  PROC DrawPart231()
    MoveL Offs(pOrigin,236.82,333.03,0.00),v40,z0,tPen\WObj:=wPaper;
    MoveL Offs(pOrigin,238.31,333.31,0.00),v40,z0,tPen\WObj:=wPaper;
    MoveL Offs(pOrigin,238.10,333.91,0.00),v40,z0,tPen\WObj:=wPaper;
    MoveL Offs(pOrigin,233.85,333.91,0.00),v40,z0,tPen\WObj:=wPaper;
    MoveL Offs(pOrigin,233.47,333.82,0.00),v40,z0,tPen\WObj:=wPaper;
    MoveL Offs(pOrigin,235.43,335.78,0.00),v40,z0,tPen\WObj:=wPaper;
    MoveL Offs(pOrigin,236.39,335.84,0.00),v40,z0,tPen\WObj:=wPaper;
    MoveL Offs(pOrigin,241.65,330.58,0.00),v40,z0,tPen\WObj:=wPaper;
    MoveL Offs(pOrigin,240.80,330.70,0.00),v40,z0,tPen\WObj:=wPaper;
    MoveL Offs(pOrigin,239.45,329.35,0.00),v40,z0,tPen\WObj:=wPaper;
    MoveL Offs(pOrigin,239.38,330.12,0.00),v40,z0,tPen\WObj:=wPaper;
    MoveL Offs(pOrigin,239.16,331.40,0.00),v40,z0,tPen\WObj:=wPaper;
    MoveL Offs(pOrigin,239.59,332.04,0.00),v40,z0,tPen\WObj:=wPaper;
    MoveL Offs(pOrigin,239.91,332.80,0.00),v40,z0,tPen\WObj:=wPaper;
    MoveL Offs(pOrigin,238.71,331.59,0.00),v40,z0,tPen\WObj:=wPaper;
    MoveL Offs(pOrigin,239.31,330.70,0.00),v40,z0,tPen\WObj:=wPaper;
    MoveL Offs(pOrigin,240.51,331.90,0.00),v40,fine,tPen\WObj:=wPaper;
    MoveL Offs(pOrigin,240.51,331.90,6.00),v60,z5,tPen\WObj:=wPaper;
    MoveL Offs(pOrigin,240.44,330.12,6.00),vTravel,z5,tPen\WObj:=wPaper;
    MoveL Offs(pOrigin,240.44,330.12,0.00),v60,z0,tPen\WObj:=wPaper;
    MoveL Offs(pOrigin,240.23,328.00,0.00),v40,z0,tPen\WObj:=wPaper;
    MoveL Offs(pOrigin,240.23,328.00,0.00),v40,z0,tPen\WObj:=wPaper;
    MoveL Offs(pOrigin,240.44,328.00,0.00),v40,z0,tPen\WObj:=wPaper;
    MoveL Offs(pOrigin,239.80,326.30,0.00),v40,z0,tPen\WObj:=wPaper;
    MoveL Offs(pOrigin,239.80,326.73,0.00),v40,z0,tPen\WObj:=wPaper;
    MoveL Offs(pOrigin,239.16,327.15,0.00),v40,z0,tPen\WObj:=wPaper;
    MoveL Offs(pOrigin,239.38,328.00,0.00),v40,z0,tPen\WObj:=wPaper;
    MoveL Offs(pOrigin,239.38,328.00,0.00),v40,z0,tPen\WObj:=wPaper;
    MoveL Offs(pOrigin,239.38,330.12,0.00),v40,z0,tPen\WObj:=wPaper;
    MoveL Offs(pOrigin,239.38,330.12,0.00),v40,z0,tPen\WObj:=wPaper;
    MoveL Offs(pOrigin,240.44,330.12,0.00),v40,z0,tPen\WObj:=wPaper;
    MoveL Offs(pOrigin,241.10,329.50,0.00),v40,z0,tPen\WObj:=wPaper;
    MoveL Offs(pOrigin,220.51,308.92,0.00),v40,z0,tPen\WObj:=wPaper;
    MoveL Offs(pOrigin,220.68,309.09,0.00),v40,z0,tPen\WObj:=wPaper;
    MoveL Offs(pOrigin,218.76,309.51,0.00),v40,z0,tPen\WObj:=wPaper;
    MoveL Offs(pOrigin,218.05,310.01,0.00),v40,z0,tPen\WObj:=wPaper;
    MoveL Offs(pOrigin,218.05,311.35,0.00),v40,z0,tPen\WObj:=wPaper;
    MoveL Offs(pOrigin,216.85,311.57,0.00),v40,z0,tPen\WObj:=wPaper;
    MoveL Offs(pOrigin,217.06,310.36,0.00),v40,z0,tPen\WObj:=wPaper;
    MoveL Offs(pOrigin,218.05,310.01,0.00),v40,z0,tPen\WObj:=wPaper;
    MoveL Offs(pOrigin,217.55,310.15,0.00),v40,z0,tPen\WObj:=wPaper;
    MoveL Offs(pOrigin,217.55,315.68,0.00),v40,z0,tPen\WObj:=wPaper;
    MoveL Offs(pOrigin,217.28,315.96,0.00),v40,z0,tPen\WObj:=wPaper;
    MoveL Offs(pOrigin,231.51,315.96,0.00),v40,z0,tPen\WObj:=wPaper;
    MoveL Offs(pOrigin,231.28,316.95,0.00),v40,z0,tPen\WObj:=wPaper;
    MoveL Offs(pOrigin,231.28,322.05,0.00),v40,z0,tPen\WObj:=wPaper;
    MoveL Offs(pOrigin,232.33,322.05,0.00),v40,z0,tPen\WObj:=wPaper;
    MoveL Offs(pOrigin,232.33,318.44,0.00),v40,z0,tPen\WObj:=wPaper;
    MoveL Offs(pOrigin,232.57,318.44,0.00),v40,z0,tPen\WObj:=wPaper;
    MoveL Offs(pOrigin,231.94,319.08,0.00),v40,z0,tPen\WObj:=wPaper;
    MoveL Offs(pOrigin,231.09,319.08,0.00),v40,z0,tPen\WObj:=wPaper;
    MoveL Offs(pOrigin,231.09,319.08,0.00),v40,z0,tPen\WObj:=wPaper;
    MoveL Offs(pOrigin,231.16,320.56,0.00),v40,z0,tPen\WObj:=wPaper;
    MoveL Offs(pOrigin,233.43,323.11,0.00),v40,z0,tPen\WObj:=wPaper;
    MoveL Offs(pOrigin,233.21,322.69,0.00),v40,z0,tPen\WObj:=wPaper;
    MoveL Offs(pOrigin,233.43,323.11,0.00),v40,z0,tPen\WObj:=wPaper;
    MoveL Offs(pOrigin,233.21,322.69,0.00),v40,z0,tPen\WObj:=wPaper;
    MoveL Offs(pOrigin,233.39,322.26,0.00),v40,z0,tPen\WObj:=wPaper;
    MoveL Offs(pOrigin,233.39,319.71,0.00),v40,fine,tPen\WObj:=wPaper;
    MoveL Offs(pOrigin,233.39,319.71,6.00),v60,z5,tPen\WObj:=wPaper;
    MoveL Offs(pOrigin,234.27,320.56,6.00),vTravel,z5,tPen\WObj:=wPaper;
    MoveL Offs(pOrigin,234.27,320.56,0.00),v60,z0,tPen\WObj:=wPaper;
    MoveL Offs(pOrigin,234.27,320.14,0.00),v40,z0,tPen\WObj:=wPaper;
    MoveL Offs(pOrigin,232.79,318.44,0.00),v40,z0,tPen\WObj:=wPaper;
    MoveL Offs(pOrigin,232.79,318.44,0.00),v40,z0,tPen\WObj:=wPaper;
    MoveL Offs(pOrigin,233.21,317.16,0.00),v40,z0,tPen\WObj:=wPaper;
    MoveL Offs(pOrigin,232.57,315.25,0.00),v40,z0,tPen\WObj:=wPaper;
    MoveL Offs(pOrigin,232.57,313.12,0.00),v40,z0,tPen\WObj:=wPaper;
    MoveL Offs(pOrigin,233.21,311.99,0.00),v40,z0,tPen\WObj:=wPaper;
    MoveL Offs(pOrigin,233.64,312.49,0.00),v40,z0,tPen\WObj:=wPaper;
    MoveL Offs(pOrigin,233.43,313.34,0.00),v40,z0,tPen\WObj:=wPaper;
    MoveL Offs(pOrigin,233.64,315.25,0.00),v40,z0,tPen\WObj:=wPaper;
    MoveL Offs(pOrigin,234.20,316.95,0.00),v40,z0,tPen\WObj:=wPaper;
    MoveL Offs(pOrigin,235.34,317.80,0.00),v40,z0,tPen\WObj:=wPaper;
    MoveL Offs(pOrigin,237.04,320.77,0.00),v40,z0,tPen\WObj:=wPaper;
    MoveL Offs(pOrigin,237.04,320.77,0.00),v40,z0,tPen\WObj:=wPaper;
    MoveL Offs(pOrigin,238.10,321.84,0.00),v40,z0,tPen\WObj:=wPaper;
    MoveL Offs(pOrigin,237.61,322.26,0.00),v40,z0,tPen\WObj:=wPaper;
    MoveL Offs(pOrigin,237.61,324.18,0.00),v40,z0,tPen\WObj:=wPaper;
    MoveL Offs(pOrigin,236.56,323.96,0.00),v40,z0,tPen\WObj:=wPaper;
    MoveL Offs(pOrigin,236.56,321.41,0.00),v40,z0,tPen\WObj:=wPaper;
    MoveL Offs(pOrigin,235.55,321.41,0.00),v40,z0,tPen\WObj:=wPaper;
    MoveL Offs(pOrigin,234.91,320.70,0.00),v40,z0,tPen\WObj:=wPaper;
    MoveL Offs(pOrigin,234.35,320.77,0.00),v40,z0,tPen\WObj:=wPaper;
    MoveL Offs(pOrigin,234.70,321.84,0.00),v40,z0,tPen\WObj:=wPaper;
    MoveL Offs(pOrigin,235.55,322.05,0.00),v40,fine,tPen\WObj:=wPaper;
    MoveL Offs(pOrigin,235.55,322.05,6.00),v60,z5,tPen\WObj:=wPaper;
    MoveL Offs(pOrigin,235.50,320.77,6.00),vTravel,z5,tPen\WObj:=wPaper;
    MoveL Offs(pOrigin,235.50,320.77,0.00),v60,z0,tPen\WObj:=wPaper;
    MoveL Offs(pOrigin,235.50,323.54,0.00),v40,z0,tPen\WObj:=wPaper;
    MoveL Offs(pOrigin,236.19,324.41,0.00),v40,z0,tPen\WObj:=wPaper;
    MoveL Offs(pOrigin,239.59,324.41,0.00),v40,z0,tPen\WObj:=wPaper;
    MoveL Offs(pOrigin,240.03,323.96,0.00),v40,z0,tPen\WObj:=wPaper;
    MoveL Offs(pOrigin,226.66,310.58,0.00),v40,fine,tPen\WObj:=wPaper;
    MoveL Offs(pOrigin,226.66,310.58,6.00),v60,z5,tPen\WObj:=wPaper;
    MoveL Offs(pOrigin,226.62,313.85,6.00),vTravel,z5,tPen\WObj:=wPaper;
    MoveL Offs(pOrigin,226.62,313.85,0.00),v60,z0,tPen\WObj:=wPaper;
    MoveL Offs(pOrigin,216.00,313.85,0.00),v40,z0,tPen\WObj:=wPaper;
    MoveL Offs(pOrigin,215.57,313.55,0.00),v40,z0,tPen\WObj:=wPaper;
    MoveL Offs(pOrigin,215.15,313.98,0.00),v40,z0,tPen\WObj:=wPaper;
    MoveL Offs(pOrigin,215.15,314.61,0.00),v40,z0,tPen\WObj:=wPaper;
    MoveL Offs(pOrigin,214.94,313.85,0.00),v40,z0,tPen\WObj:=wPaper;
    MoveL Offs(pOrigin,213.24,313.85,0.00),v40,z0,tPen\WObj:=wPaper;
    MoveL Offs(pOrigin,212.81,314.40,0.00),v40,z0,tPen\WObj:=wPaper;
    MoveL Offs(pOrigin,212.60,314.83,0.00),v40,z0,tPen\WObj:=wPaper;
    MoveL Offs(pOrigin,212.81,314.40,0.00),v40,z0,tPen\WObj:=wPaper;
    MoveL Offs(pOrigin,212.81,314.90,0.00),v40,z0,tPen\WObj:=wPaper;
    MoveL Offs(pOrigin,214.30,314.90,0.00),v40,z0,tPen\WObj:=wPaper;
    MoveL Offs(pOrigin,213.88,315.96,0.00),v40,z0,tPen\WObj:=wPaper;
    MoveL Offs(pOrigin,212.60,315.96,0.00),v40,z0,tPen\WObj:=wPaper;
    MoveL Offs(pOrigin,211.96,315.67,0.00),v40,z0,tPen\WObj:=wPaper;
    MoveL Offs(pOrigin,212.88,314.61,0.00),v40,z0,tPen\WObj:=wPaper;
    MoveL Offs(pOrigin,213.24,313.55,0.00),v40,z0,tPen\WObj:=wPaper;
    MoveL Offs(pOrigin,213.02,313.12,0.00),v40,z0,tPen\WObj:=wPaper;
    MoveL Offs(pOrigin,212.18,312.79,0.00),v40,z0,tPen\WObj:=wPaper;
    MoveL Offs(pOrigin,224.08,312.79,0.00),v40,fine,tPen\WObj:=wPaper;
    MoveL Offs(pOrigin,224.08,312.79,6.00),v60,z5,tPen\WObj:=wPaper;
    MoveL Offs(pOrigin,224.94,314.40,6.00),vTravel,z5,tPen\WObj:=wPaper;
    MoveL Offs(pOrigin,224.94,314.40,0.00),v60,z0,tPen\WObj:=wPaper;
    MoveL Offs(pOrigin,224.94,319.92,0.00),v40,z0,tPen\WObj:=wPaper;
  ENDPROC

  PROC DrawPart232()
    MoveL Offs(pOrigin,223.89,320.35,0.00),v40,z0,tPen\WObj:=wPaper;
    MoveL Offs(pOrigin,223.89,315.68,0.00),v40,z0,tPen\WObj:=wPaper;
    MoveL Offs(pOrigin,224.29,316.10,0.00),v40,z0,tPen\WObj:=wPaper;
    MoveL Offs(pOrigin,224.07,314.61,0.00),v40,z0,tPen\WObj:=wPaper;
    MoveL Offs(pOrigin,224.64,313.76,0.00),v40,z0,tPen\WObj:=wPaper;
    MoveL Offs(pOrigin,224.64,312.49,0.00),v40,z0,tPen\WObj:=wPaper;
    MoveL Offs(pOrigin,225.42,310.79,0.00),v40,z0,tPen\WObj:=wPaper;
    MoveL Offs(pOrigin,227.48,310.65,0.00),v40,z0,tPen\WObj:=wPaper;
    MoveL Offs(pOrigin,226.84,313.12,0.00),v40,z0,tPen\WObj:=wPaper;
    MoveL Offs(pOrigin,226.84,314.40,0.00),v40,z0,tPen\WObj:=wPaper;
    MoveL Offs(pOrigin,228.54,318.23,0.00),v40,fine,tPen\WObj:=wPaper;
    MoveL Offs(pOrigin,228.54,318.23,6.00),v60,z5,tPen\WObj:=wPaper;
    MoveL Offs(pOrigin,228.96,316.74,6.00),vTravel,z5,tPen\WObj:=wPaper;
    MoveL Offs(pOrigin,228.96,316.74,0.00),v60,z0,tPen\WObj:=wPaper;
    MoveL Offs(pOrigin,229.81,316.74,0.00),v40,z0,tPen\WObj:=wPaper;
    MoveL Offs(pOrigin,230.66,318.01,0.00),v40,z0,tPen\WObj:=wPaper;
    MoveL Offs(pOrigin,230.66,318.01,0.00),v40,z0,tPen\WObj:=wPaper;
    MoveL Offs(pOrigin,231.09,319.08,0.00),v40,fine,tPen\WObj:=wPaper;
    MoveL Offs(pOrigin,231.09,319.08,6.00),v60,z5,tPen\WObj:=wPaper;
    MoveL Offs(pOrigin,231.30,317.80,6.00),vTravel,z5,tPen\WObj:=wPaper;
    MoveL Offs(pOrigin,231.30,317.80,0.00),v60,z0,tPen\WObj:=wPaper;
    MoveL Offs(pOrigin,231.94,317.80,0.00),v40,z0,tPen\WObj:=wPaper;
    MoveL Offs(pOrigin,232.57,318.44,0.00),v40,z0,tPen\WObj:=wPaper;
    MoveL Offs(pOrigin,232.79,318.44,0.00),v40,z0,tPen\WObj:=wPaper;
    MoveL Offs(pOrigin,232.15,317.80,0.00),v40,z0,tPen\WObj:=wPaper;
    MoveL Offs(pOrigin,232.15,317.80,0.00),v40,z0,tPen\WObj:=wPaper;
    MoveL Offs(pOrigin,231.51,314.61,0.00),v40,z0,tPen\WObj:=wPaper;
    MoveL Offs(pOrigin,230.88,313.76,0.00),v40,z0,tPen\WObj:=wPaper;
    MoveL Offs(pOrigin,230.88,313.76,0.00),v40,z0,tPen\WObj:=wPaper;
    MoveL Offs(pOrigin,230.80,312.27,0.00),v40,z0,tPen\WObj:=wPaper;
    MoveL Offs(pOrigin,229.25,312.91,0.00),v40,z0,tPen\WObj:=wPaper;
    MoveL Offs(pOrigin,228.96,316.74,0.00),v40,fine,tPen\WObj:=wPaper;
    MoveL Offs(pOrigin,228.96,316.74,6.00),v60,z5,tPen\WObj:=wPaper;
    MoveL Offs(pOrigin,230.45,316.10,6.00),vTravel,z5,tPen\WObj:=wPaper;
    MoveL Offs(pOrigin,230.45,316.10,0.00),v60,z0,tPen\WObj:=wPaper;
    MoveL Offs(pOrigin,230.45,314.19,0.00),v40,z0,tPen\WObj:=wPaper;
    MoveL Offs(pOrigin,230.88,313.76,0.00),v40,z0,tPen\WObj:=wPaper;
    MoveL Offs(pOrigin,230.88,313.85,0.00),v40,z0,tPen\WObj:=wPaper;
    MoveL Offs(pOrigin,227.90,313.85,0.00),v40,fine,tPen\WObj:=wPaper;
    MoveL Offs(pOrigin,227.90,313.85,6.00),v60,z5,tPen\WObj:=wPaper;
    MoveL Offs(pOrigin,229.17,315.04,6.00),vTravel,z5,tPen\WObj:=wPaper;
    MoveL Offs(pOrigin,229.17,315.04,0.00),v60,z0,tPen\WObj:=wPaper;
    MoveL Offs(pOrigin,229.17,321.62,0.00),v40,z0,tPen\WObj:=wPaper;
    MoveL Offs(pOrigin,229.39,322.30,0.00),v40,z0,tPen\WObj:=wPaper;
    MoveL Offs(pOrigin,247.66,322.30,0.00),v40,z0,tPen\WObj:=wPaper;
    MoveL Offs(pOrigin,248.17,321.41,0.00),v40,z0,tPen\WObj:=wPaper;
    MoveL Offs(pOrigin,248.17,319.29,0.00),v40,z0,tPen\WObj:=wPaper;
    MoveL Offs(pOrigin,248.94,319.08,0.00),v40,z0,tPen\WObj:=wPaper;
    MoveL Offs(pOrigin,249.79,318.65,0.00),v40,z0,tPen\WObj:=wPaper;
    MoveL Offs(pOrigin,249.79,318.65,0.00),v40,z0,tPen\WObj:=wPaper;
    MoveL Offs(pOrigin,249.50,317.16,0.00),v40,z0,tPen\WObj:=wPaper;
    MoveL Offs(pOrigin,248.02,315.89,0.00),v40,z0,tPen\WObj:=wPaper;
    MoveL Offs(pOrigin,247.17,313.12,0.00),v40,z0,tPen\WObj:=wPaper;
    MoveL Offs(pOrigin,246.81,312.84,0.00),v40,z0,tPen\WObj:=wPaper;
    MoveL Offs(pOrigin,246.39,313.34,0.00),v40,z0,tPen\WObj:=wPaper;
    MoveL Offs(pOrigin,246.39,314.40,0.00),v40,z0,tPen\WObj:=wPaper;
    MoveL Offs(pOrigin,247.02,317.16,0.00),v40,z0,tPen\WObj:=wPaper;
    MoveL Offs(pOrigin,247.02,317.16,0.00),v40,z0,tPen\WObj:=wPaper;
    MoveL Offs(pOrigin,247.45,318.86,0.00),v40,z0,tPen\WObj:=wPaper;
    MoveL Offs(pOrigin,247.45,318.86,0.00),v40,z0,tPen\WObj:=wPaper;
    MoveL Offs(pOrigin,245.75,318.44,0.00),v40,z0,tPen\WObj:=wPaper;
    MoveL Offs(pOrigin,244.05,318.44,0.00),v40,z0,tPen\WObj:=wPaper;
    MoveL Offs(pOrigin,244.05,318.44,0.00),v40,z0,tPen\WObj:=wPaper;
    MoveL Offs(pOrigin,244.26,319.50,0.00),v40,z0,tPen\WObj:=wPaper;
    MoveL Offs(pOrigin,245.11,320.56,0.00),v40,z0,tPen\WObj:=wPaper;
    MoveL Offs(pOrigin,245.11,320.56,0.00),v40,z0,tPen\WObj:=wPaper;
    MoveL Offs(pOrigin,244.26,322.05,0.00),v40,fine,tPen\WObj:=wPaper;
    MoveL Offs(pOrigin,244.26,322.05,6.00),v60,z5,tPen\WObj:=wPaper;
    MoveL Offs(pOrigin,245.54,323.35,6.00),vTravel,z5,tPen\WObj:=wPaper;
    MoveL Offs(pOrigin,245.54,323.35,0.00),v60,z0,tPen\WObj:=wPaper;
    MoveL Offs(pOrigin,241.29,323.35,0.00),v40,z0,tPen\WObj:=wPaper;
    MoveL Offs(pOrigin,241.84,323.54,0.00),v40,z0,tPen\WObj:=wPaper;
    MoveL Offs(pOrigin,241.84,322.05,0.00),v40,fine,tPen\WObj:=wPaper;
    MoveL Offs(pOrigin,241.84,322.05,6.00),v60,z5,tPen\WObj:=wPaper;
    MoveL Offs(pOrigin,240.78,322.69,6.00),vTravel,z5,tPen\WObj:=wPaper;
    MoveL Offs(pOrigin,240.78,322.69,0.00),v60,z0,tPen\WObj:=wPaper;
    MoveL Offs(pOrigin,240.78,320.99,0.00),v40,z0,tPen\WObj:=wPaper;
    MoveL Offs(pOrigin,240.44,320.14,0.00),v40,z0,tPen\WObj:=wPaper;
    MoveL Offs(pOrigin,241.29,320.99,0.00),v40,z0,tPen\WObj:=wPaper;
    MoveL Offs(pOrigin,240.44,320.14,0.00),v40,z0,tPen\WObj:=wPaper;
    MoveL Offs(pOrigin,240.78,319.71,0.00),v40,z0,tPen\WObj:=wPaper;
    MoveL Offs(pOrigin,240.78,318.22,0.00),v40,z0,tPen\WObj:=wPaper;
    MoveL Offs(pOrigin,241.84,318.65,0.00),v40,z0,tPen\WObj:=wPaper;
    MoveL Offs(pOrigin,241.84,320.56,0.00),v40,fine,tPen\WObj:=wPaper;
    MoveL Offs(pOrigin,241.84,320.56,6.00),v60,z5,tPen\WObj:=wPaper;
    MoveL Offs(pOrigin,239.73,319.92,6.00),vTravel,z5,tPen\WObj:=wPaper;
    MoveL Offs(pOrigin,239.73,319.92,0.00),v60,z0,tPen\WObj:=wPaper;
    MoveL Offs(pOrigin,239.73,322.05,0.00),v40,fine,tPen\WObj:=wPaper;
    MoveL Offs(pOrigin,239.73,322.05,6.00),v60,z5,tPen\WObj:=wPaper;
    MoveL Offs(pOrigin,238.67,321.41,6.00),vTravel,z5,tPen\WObj:=wPaper;
    MoveL Offs(pOrigin,238.67,321.41,0.00),v60,z0,tPen\WObj:=wPaper;
    MoveL Offs(pOrigin,238.67,319.08,0.00),v40,fine,tPen\WObj:=wPaper;
    MoveL Offs(pOrigin,238.67,319.08,6.00),v60,z5,tPen\WObj:=wPaper;
    MoveL Offs(pOrigin,237.61,320.35,6.00),vTravel,z5,tPen\WObj:=wPaper;
    MoveL Offs(pOrigin,237.61,320.35,0.00),v60,z0,tPen\WObj:=wPaper;
    MoveL Offs(pOrigin,237.61,317.80,0.00),v40,fine,tPen\WObj:=wPaper;
    MoveL Offs(pOrigin,237.61,317.80,6.00),v60,z5,tPen\WObj:=wPaper;
    MoveL Offs(pOrigin,236.82,315.96,6.00),vTravel,z5,tPen\WObj:=wPaper;
    MoveL Offs(pOrigin,236.82,315.96,0.00),v60,z0,tPen\WObj:=wPaper;
    MoveL Offs(pOrigin,235.34,315.96,0.00),v40,fine,tPen\WObj:=wPaper;
    MoveL Offs(pOrigin,235.34,315.96,6.00),v60,z5,tPen\WObj:=wPaper;
    MoveL Offs(pOrigin,235.12,317.38,6.00),vTravel,z5,tPen\WObj:=wPaper;
    MoveL Offs(pOrigin,235.12,317.38,0.00),v60,z0,tPen\WObj:=wPaper;
    MoveL Offs(pOrigin,234.70,315.46,0.00),v40,z0,tPen\WObj:=wPaper;
    MoveL Offs(pOrigin,234.70,312.49,0.00),v40,z0,tPen\WObj:=wPaper;
    MoveL Offs(pOrigin,234.98,311.71,0.00),v40,z0,tPen\WObj:=wPaper;
    MoveL Offs(pOrigin,235.55,311.42,0.00),v40,z0,tPen\WObj:=wPaper;
    MoveL Offs(pOrigin,235.55,311.42,0.00),v40,z0,tPen\WObj:=wPaper;
    MoveL Offs(pOrigin,235.76,310.79,0.00),v40,z0,tPen\WObj:=wPaper;
    MoveL Offs(pOrigin,237.25,309.51,0.00),v40,z0,tPen\WObj:=wPaper;
    MoveL Offs(pOrigin,237.81,310.52,0.00),v40,z0,tPen\WObj:=wPaper;
    MoveL Offs(pOrigin,213.02,335.31,0.00),v40,z0,tPen\WObj:=wPaper;
    MoveL Offs(pOrigin,211.97,334.86,0.00),v40,z0,tPen\WObj:=wPaper;
    MoveL Offs(pOrigin,236.46,310.37,0.00),v40,fine,tPen\WObj:=wPaper;
    MoveL Offs(pOrigin,236.46,310.37,6.00),v60,z5,tPen\WObj:=wPaper;
    MoveL Offs(pOrigin,234.76,312.71,6.00),vTravel,z5,tPen\WObj:=wPaper;
    MoveL Offs(pOrigin,234.76,312.71,0.00),v60,z0,tPen\WObj:=wPaper;
    MoveL Offs(pOrigin,246.78,324.73,0.00),v40,fine,tPen\WObj:=wPaper;
    MoveL Offs(pOrigin,246.78,324.73,6.00),v60,z5,tPen\WObj:=wPaper;
    MoveL Offs(pOrigin,245.14,327.57,6.00),vTravel,z5,tPen\WObj:=wPaper;
  ENDPROC

  PROC DrawPart233()
    MoveL Offs(pOrigin,245.14,327.57,0.00),v60,z0,tPen\WObj:=wPaper;
    MoveL Offs(pOrigin,229.81,312.24,0.00),v40,fine,tPen\WObj:=wPaper;
    MoveL Offs(pOrigin,229.81,312.24,6.00),v60,z5,tPen\WObj:=wPaper;
    MoveL Offs(pOrigin,230.22,314.40,6.00),vTravel,z5,tPen\WObj:=wPaper;
    MoveL Offs(pOrigin,230.22,314.40,0.00),v60,z0,tPen\WObj:=wPaper;
    MoveL Offs(pOrigin,230.22,322.05,0.00),v40,fine,tPen\WObj:=wPaper;
    MoveL Offs(pOrigin,230.22,322.05,6.00),v60,z5,tPen\WObj:=wPaper;
    MoveL Offs(pOrigin,228.32,322.26,6.00),vTravel,z5,tPen\WObj:=wPaper;
    MoveL Offs(pOrigin,228.32,322.26,0.00),v60,z0,tPen\WObj:=wPaper;
    MoveL Offs(pOrigin,228.54,325.66,0.00),v40,z0,tPen\WObj:=wPaper;
    MoveL Offs(pOrigin,227.90,326.30,0.00),v40,fine,tPen\WObj:=wPaper;
    MoveL Offs(pOrigin,227.90,326.30,6.00),v60,z5,tPen\WObj:=wPaper;
    MoveL Offs(pOrigin,229.53,326.27,6.00),vTravel,z5,tPen\WObj:=wPaper;
    MoveL Offs(pOrigin,229.53,326.27,0.00),v60,z0,tPen\WObj:=wPaper;
    MoveL Offs(pOrigin,244.25,311.55,0.00),v40,z0,tPen\WObj:=wPaper;
    MoveL Offs(pOrigin,245.11,311.64,0.00),v40,z0,tPen\WObj:=wPaper;
    MoveL Offs(pOrigin,245.11,314.19,0.00),v40,z0,tPen\WObj:=wPaper;
    MoveL Offs(pOrigin,245.68,315.89,0.00),v40,z0,tPen\WObj:=wPaper;
    MoveL Offs(pOrigin,246.39,316.95,0.00),v40,z0,tPen\WObj:=wPaper;
    MoveL Offs(pOrigin,247.02,317.16,0.00),v40,z0,tPen\WObj:=wPaper;
    MoveL Offs(pOrigin,246.18,317.02,0.00),v40,z0,tPen\WObj:=wPaper;
    MoveL Offs(pOrigin,244.48,317.02,0.00),v40,z0,tPen\WObj:=wPaper;
    MoveL Offs(pOrigin,245.01,316.95,0.00),v40,z0,tPen\WObj:=wPaper;
    MoveL Offs(pOrigin,245.01,319.50,0.00),v40,z0,tPen\WObj:=wPaper;
    MoveL Offs(pOrigin,244.69,319.92,0.00),v40,z0,tPen\WObj:=wPaper;
    MoveL Offs(pOrigin,245.54,320.70,0.00),v40,z0,tPen\WObj:=wPaper;
    MoveL Offs(pOrigin,247.24,321.41,0.00),v40,z0,tPen\WObj:=wPaper;
    MoveL Offs(pOrigin,248.73,323.47,0.00),v40,z0,tPen\WObj:=wPaper;
    MoveL Offs(pOrigin,250.43,324.17,0.00),v40,z0,tPen\WObj:=wPaper;
    MoveL Offs(pOrigin,252.27,326.16,0.00),v40,z0,tPen\WObj:=wPaper;
    MoveL Offs(pOrigin,252.55,329.06,0.00),v40,z0,tPen\WObj:=wPaper;
    MoveL Offs(pOrigin,251.77,331.19,0.00),v40,z0,tPen\WObj:=wPaper;
    MoveL Offs(pOrigin,250.85,331.61,0.00),v40,z0,tPen\WObj:=wPaper;
    MoveL Offs(pOrigin,249.94,330.88,0.00),v40,z0,tPen\WObj:=wPaper;
    MoveL Offs(pOrigin,251.89,332.83,0.00),v40,z0,tPen\WObj:=wPaper;
    MoveL Offs(pOrigin,251.91,333.10,0.00),v40,z0,tPen\WObj:=wPaper;
    MoveL Offs(pOrigin,252.12,332.67,0.00),v40,z0,tPen\WObj:=wPaper;
    MoveL Offs(pOrigin,251.91,333.10,0.00),v40,z0,tPen\WObj:=wPaper;
    MoveL Offs(pOrigin,251.27,333.74,0.00),v40,z0,tPen\WObj:=wPaper;
    MoveL Offs(pOrigin,251.49,333.31,0.00),v40,z0,tPen\WObj:=wPaper;
    MoveL Offs(pOrigin,251.27,333.74,0.00),v40,z0,tPen\WObj:=wPaper;
    MoveL Offs(pOrigin,251.00,333.43,0.00),v40,z0,tPen\WObj:=wPaper;
    MoveL Offs(pOrigin,249.65,332.08,0.00),v40,z0,tPen\WObj:=wPaper;
    MoveL Offs(pOrigin,249.05,332.97,0.00),v40,z0,tPen\WObj:=wPaper;
    MoveL Offs(pOrigin,250.25,334.18,0.00),v40,z0,tPen\WObj:=wPaper;
    MoveL Offs(pOrigin,250.64,334.38,0.00),v40,z0,tPen\WObj:=wPaper;
    MoveL Offs(pOrigin,250.85,333.95,0.00),v40,z0,tPen\WObj:=wPaper;
    MoveL Offs(pOrigin,250.64,334.38,0.00),v40,fine,tPen\WObj:=wPaper;
    MoveL Offs(pOrigin,250.64,334.38,6.00),v60,z5,tPen\WObj:=wPaper;
    MoveL Offs(pOrigin,249.15,333.95,6.00),vTravel,z5,tPen\WObj:=wPaper;
    MoveL Offs(pOrigin,249.15,333.95,0.00),v60,z0,tPen\WObj:=wPaper;
    MoveL Offs(pOrigin,247.45,334.23,0.00),v40,z0,tPen\WObj:=wPaper;
    MoveL Offs(pOrigin,246.39,335.23,0.00),v40,fine,tPen\WObj:=wPaper;
    MoveL Offs(pOrigin,246.39,335.23,6.00),v60,z5,tPen\WObj:=wPaper;
    MoveL Offs(pOrigin,244.69,337.08,6.00),vTravel,z5,tPen\WObj:=wPaper;
    MoveL Offs(pOrigin,244.69,337.08,0.00),v60,z0,tPen\WObj:=wPaper;
    MoveL Offs(pOrigin,239.38,337.08,0.00),v40,z0,tPen\WObj:=wPaper;
    MoveL Offs(pOrigin,239.32,336.69,0.00),v40,z0,tPen\WObj:=wPaper;
    MoveL Offs(pOrigin,242.33,339.69,0.00),v40,z0,tPen\WObj:=wPaper;
    MoveL Offs(pOrigin,242.67,340.01,0.00),v40,z0,tPen\WObj:=wPaper;
    MoveL Offs(pOrigin,254.08,328.59,0.00),v40,z0,tPen\WObj:=wPaper;
    MoveL Offs(pOrigin,253.53,328.49,0.00),v40,z0,tPen\WObj:=wPaper;
    MoveL Offs(pOrigin,252.63,327.59,0.00),v40,z0,tPen\WObj:=wPaper;
    MoveL Offs(pOrigin,253.52,326.99,0.00),v40,z0,tPen\WObj:=wPaper;
    MoveL Offs(pOrigin,240.90,314.37,0.00),v40,fine,tPen\WObj:=wPaper;
    MoveL Offs(pOrigin,240.90,314.37,6.00),v60,z5,tPen\WObj:=wPaper;
    MoveL Offs(pOrigin,241.20,313.18,6.00),vTravel,z5,tPen\WObj:=wPaper;
    MoveL Offs(pOrigin,241.20,313.18,0.00),v60,z0,tPen\WObj:=wPaper;
    MoveL Offs(pOrigin,242.55,314.53,0.00),v40,fine,tPen\WObj:=wPaper;
    MoveL Offs(pOrigin,242.55,314.53,6.00),v60,z5,tPen\WObj:=wPaper;
    MoveL Offs(pOrigin,243.75,314.23,6.00),vTravel,z5,tPen\WObj:=wPaper;
    MoveL Offs(pOrigin,243.75,314.23,0.00),v60,z0,tPen\WObj:=wPaper;
    MoveL Offs(pOrigin,256.67,327.15,0.00),v40,z0,tPen\WObj:=wPaper;
    MoveL Offs(pOrigin,255.62,327.60,0.00),v40,z0,tPen\WObj:=wPaper;
    MoveL Offs(pOrigin,256.37,328.35,0.00),v40,fine,tPen\WObj:=wPaper;
    MoveL Offs(pOrigin,256.37,328.35,6.00),v60,z5,tPen\WObj:=wPaper;
    MoveL Offs(pOrigin,255.13,329.04,6.00),vTravel,z5,tPen\WObj:=wPaper;
    MoveL Offs(pOrigin,255.13,329.04,0.00),v60,z0,tPen\WObj:=wPaper;
    MoveL Offs(pOrigin,299.01,285.16,0.00),v40,fine,tPen\WObj:=wPaper;
    MoveL Offs(pOrigin,299.01,285.16,6.00),v60,z5,tPen\WObj:=wPaper;
    MoveL Offs(pOrigin,299.01,283.67,6.00),vTravel,z5,tPen\WObj:=wPaper;
    MoveL Offs(pOrigin,299.01,283.67,0.00),v60,z0,tPen\WObj:=wPaper;
    MoveL Offs(pOrigin,254.99,327.69,0.00),v40,fine,tPen\WObj:=wPaper;
    MoveL Offs(pOrigin,254.99,327.69,6.00),v60,z5,tPen\WObj:=wPaper;
    MoveL Offs(pOrigin,254.98,330.69,6.00),vTravel,z5,tPen\WObj:=wPaper;
    MoveL Offs(pOrigin,254.98,330.69,0.00),v60,z0,tPen\WObj:=wPaper;
    MoveL Offs(pOrigin,260.39,325.28,0.00),v40,z0,tPen\WObj:=wPaper;
    MoveL Offs(pOrigin,260.11,326.12,0.00),v40,z0,tPen\WObj:=wPaper;
    MoveL Offs(pOrigin,248.84,314.85,0.00),v40,fine,tPen\WObj:=wPaper;
    MoveL Offs(pOrigin,248.84,314.85,6.00),v60,z5,tPen\WObj:=wPaper;
    MoveL Offs(pOrigin,247.20,314.69,6.00),vTravel,z5,tPen\WObj:=wPaper;
    MoveL Offs(pOrigin,247.20,314.69,0.00),v60,z0,tPen\WObj:=wPaper;
    MoveL Offs(pOrigin,260.42,327.91,0.00),v40,z0,tPen\WObj:=wPaper;
    MoveL Offs(pOrigin,260.98,327.67,0.00),v40,z0,tPen\WObj:=wPaper;
    MoveL Offs(pOrigin,248.81,339.84,0.00),v40,fine,tPen\WObj:=wPaper;
    MoveL Offs(pOrigin,248.81,339.84,6.00),v60,z5,tPen\WObj:=wPaper;
    MoveL Offs(pOrigin,248.30,338.14,6.00),vTravel,z5,tPen\WObj:=wPaper;
    MoveL Offs(pOrigin,248.30,338.14,0.00),v60,z0,tPen\WObj:=wPaper;
    MoveL Offs(pOrigin,255.95,338.14,0.00),v40,z0,tPen\WObj:=wPaper;
    MoveL Offs(pOrigin,256.26,338.69,0.00),v40,z0,tPen\WObj:=wPaper;
    MoveL Offs(pOrigin,253.40,335.83,0.00),v40,z0,tPen\WObj:=wPaper;
    MoveL Offs(pOrigin,253.61,335.65,0.00),v40,z0,tPen\WObj:=wPaper;
    MoveL Offs(pOrigin,253.40,335.86,0.00),v40,z0,tPen\WObj:=wPaper;
    MoveL Offs(pOrigin,253.61,335.44,0.00),v40,z0,tPen\WObj:=wPaper;
    MoveL Offs(pOrigin,254.25,335.44,0.00),v40,z0,tPen\WObj:=wPaper;
    MoveL Offs(pOrigin,254.25,335.44,0.00),v40,z0,tPen\WObj:=wPaper;
    MoveL Offs(pOrigin,255.10,334.52,0.00),v40,z0,tPen\WObj:=wPaper;
    MoveL Offs(pOrigin,255.95,334.45,0.00),v40,z0,tPen\WObj:=wPaper;
    MoveL Offs(pOrigin,255.52,335.65,0.00),v40,z0,tPen\WObj:=wPaper;
    MoveL Offs(pOrigin,254.68,336.08,0.00),v40,z0,tPen\WObj:=wPaper;
    MoveL Offs(pOrigin,254.68,336.08,0.00),v40,z0,tPen\WObj:=wPaper;
    MoveL Offs(pOrigin,254.04,337.14,0.00),v40,z0,tPen\WObj:=wPaper;
    MoveL Offs(pOrigin,254.04,337.14,0.00),v40,z0,tPen\WObj:=wPaper;
    MoveL Offs(pOrigin,254.89,337.63,0.00),v40,z0,tPen\WObj:=wPaper;
    MoveL Offs(pOrigin,257.65,336.29,0.00),v40,z0,tPen\WObj:=wPaper;
    MoveL Offs(pOrigin,257.01,336.02,0.00),v40,z0,tPen\WObj:=wPaper;
    MoveL Offs(pOrigin,254.04,336.02,0.00),v40,z0,tPen\WObj:=wPaper;
    MoveL Offs(pOrigin,254.51,336.29,0.00),v40,z0,tPen\WObj:=wPaper;
    MoveL Offs(pOrigin,254.51,338.20,0.00),v40,z0,tPen\WObj:=wPaper;
    MoveL Offs(pOrigin,255.06,338.98,0.00),v40,z0,tPen\WObj:=wPaper;
  ENDPROC

  PROC DrawPart234()
    MoveL Offs(pOrigin,252.66,336.58,0.00),v40,z0,tPen\WObj:=wPaper;
    MoveL Offs(pOrigin,252.76,337.08,0.00),v40,z0,tPen\WObj:=wPaper;
    MoveL Offs(pOrigin,258.92,337.08,0.00),v40,z0,tPen\WObj:=wPaper;
    MoveL Offs(pOrigin,259.14,337.56,0.00),v40,z0,tPen\WObj:=wPaper;
    MoveL Offs(pOrigin,258.50,338.06,0.00),v40,z0,tPen\WObj:=wPaper;
    MoveL Offs(pOrigin,255.52,339.05,0.00),v40,z0,tPen\WObj:=wPaper;
    MoveL Offs(pOrigin,252.12,339.69,0.00),v40,z0,tPen\WObj:=wPaper;
    MoveL Offs(pOrigin,242.77,339.90,0.00),v40,z0,tPen\WObj:=wPaper;
    MoveL Offs(pOrigin,241.93,339.62,0.00),v40,z0,tPen\WObj:=wPaper;
    MoveL Offs(pOrigin,241.71,339.05,0.00),v40,z0,tPen\WObj:=wPaper;
    MoveL Offs(pOrigin,241.71,339.69,0.00),v40,z0,tPen\WObj:=wPaper;
    MoveL Offs(pOrigin,237.68,339.90,0.00),v40,z0,tPen\WObj:=wPaper;
    MoveL Offs(pOrigin,235.76,340.33,0.00),v40,z0,tPen\WObj:=wPaper;
    MoveL Offs(pOrigin,230.88,340.33,0.00),v40,z0,tPen\WObj:=wPaper;
    MoveL Offs(pOrigin,227.48,339.69,0.00),v40,z0,tPen\WObj:=wPaper;
    MoveL Offs(pOrigin,218.55,336.50,0.00),v40,z0,tPen\WObj:=wPaper;
    MoveL Offs(pOrigin,213.02,335.08,0.00),v40,z0,tPen\WObj:=wPaper;
    MoveL Offs(pOrigin,208.56,332.89,0.00),v40,z0,tPen\WObj:=wPaper;
    MoveL Offs(pOrigin,204.95,329.49,0.00),v40,z0,tPen\WObj:=wPaper;
    MoveL Offs(pOrigin,203.32,326.94,0.00),v40,z0,tPen\WObj:=wPaper;
    MoveL Offs(pOrigin,203.46,326.58,0.00),v40,z0,tPen\WObj:=wPaper;
    MoveL Offs(pOrigin,204.52,326.51,0.00),v40,z0,tPen\WObj:=wPaper;
    MoveL Offs(pOrigin,204.52,326.51,0.00),v40,z0,tPen\WObj:=wPaper;
    MoveL Offs(pOrigin,204.24,325.31,0.00),v40,z0,tPen\WObj:=wPaper;
    MoveL Offs(pOrigin,203.04,325.02,0.00),v40,z0,tPen\WObj:=wPaper;
    MoveL Offs(pOrigin,202.11,325.31,0.00),v40,z0,tPen\WObj:=wPaper;
    MoveL Offs(pOrigin,207.82,319.60,0.00),v40,fine,tPen\WObj:=wPaper;
    MoveL Offs(pOrigin,207.82,319.60,6.00),v60,z5,tPen\WObj:=wPaper;
    MoveL Offs(pOrigin,210.69,320.18,6.00),vTravel,z5,tPen\WObj:=wPaper;
    MoveL Offs(pOrigin,210.69,320.18,0.00),v60,z0,tPen\WObj:=wPaper;
    MoveL Offs(pOrigin,211.96,320.18,0.00),v40,z0,tPen\WObj:=wPaper;
    MoveL Offs(pOrigin,211.75,320.56,0.00),v40,z0,tPen\WObj:=wPaper;
    MoveL Offs(pOrigin,211.96,320.99,0.00),v40,z0,tPen\WObj:=wPaper;
    MoveL Offs(pOrigin,211.75,320.56,0.00),v40,z0,tPen\WObj:=wPaper;
    MoveL Offs(pOrigin,211.96,320.99,0.00),v40,z0,tPen\WObj:=wPaper;
    MoveL Offs(pOrigin,211.75,321.34,0.00),v40,z0,tPen\WObj:=wPaper;
    MoveL Offs(pOrigin,208.77,322.69,0.00),v40,z0,tPen\WObj:=wPaper;
    MoveL Offs(pOrigin,205.16,322.90,0.00),v40,fine,tPen\WObj:=wPaper;
    MoveL Offs(pOrigin,205.16,322.90,6.00),v60,z5,tPen\WObj:=wPaper;
    MoveL Offs(pOrigin,203.94,326.69,6.00),vTravel,z5,tPen\WObj:=wPaper;
    MoveL Offs(pOrigin,203.94,326.69,0.00),v60,z0,tPen\WObj:=wPaper;
    MoveL Offs(pOrigin,205.29,328.05,0.00),v40,z0,tPen\WObj:=wPaper;
    MoveL Offs(pOrigin,205.59,328.64,0.00),v40,z0,tPen\WObj:=wPaper;
    MoveL Offs(pOrigin,205.80,329.06,0.00),v40,z0,tPen\WObj:=wPaper;
    MoveL Offs(pOrigin,205.59,328.64,0.00),v40,z0,tPen\WObj:=wPaper;
    MoveL Offs(pOrigin,206.01,329.27,0.00),v40,z0,tPen\WObj:=wPaper;
    MoveL Offs(pOrigin,207.07,330.34,0.00),v40,z0,tPen\WObj:=wPaper;
    MoveL Offs(pOrigin,206.01,329.27,0.00),v40,fine,tPen\WObj:=wPaper;
    MoveL Offs(pOrigin,206.01,329.27,6.00),v60,z5,tPen\WObj:=wPaper;
    MoveL Offs(pOrigin,207.29,328.85,6.00),vTravel,z5,tPen\WObj:=wPaper;
    MoveL Offs(pOrigin,207.29,328.85,0.00),v60,z0,tPen\WObj:=wPaper;
    MoveL Offs(pOrigin,208.14,329.49,0.00),v40,z0,tPen\WObj:=wPaper;
    MoveL Offs(pOrigin,207.29,328.85,0.00),v40,fine,tPen\WObj:=wPaper;
    MoveL Offs(pOrigin,207.29,328.85,6.00),v60,z5,tPen\WObj:=wPaper;
    MoveL Offs(pOrigin,207.50,327.58,6.00),vTravel,z5,tPen\WObj:=wPaper;
    MoveL Offs(pOrigin,207.50,327.58,0.00),v60,z0,tPen\WObj:=wPaper;
    MoveL Offs(pOrigin,218.76,327.58,0.00),v40,z0,tPen\WObj:=wPaper;
    MoveL Offs(pOrigin,219.19,327.36,0.00),v40,z0,tPen\WObj:=wPaper;
    MoveL Offs(pOrigin,218.34,326.73,0.00),v40,z0,tPen\WObj:=wPaper;
    MoveL Offs(pOrigin,218.76,326.73,0.00),v40,z0,tPen\WObj:=wPaper;
    MoveL Offs(pOrigin,219.61,327.36,0.00),v40,z0,tPen\WObj:=wPaper;
    MoveL Offs(pOrigin,220.68,327.29,0.00),v40,z0,tPen\WObj:=wPaper;
    MoveL Offs(pOrigin,221.88,326.30,0.00),v40,z0,tPen\WObj:=wPaper;
    MoveL Offs(pOrigin,221.95,325.66,0.00),v40,z0,tPen\WObj:=wPaper;
    MoveL Offs(pOrigin,221.74,326.30,0.00),v40,z0,tPen\WObj:=wPaper;
    MoveL Offs(pOrigin,221.52,326.73,0.00),v40,z0,tPen\WObj:=wPaper;
    MoveL Offs(pOrigin,221.74,326.30,0.00),v40,fine,tPen\WObj:=wPaper;
    MoveL Offs(pOrigin,221.74,326.30,6.00),v60,z5,tPen\WObj:=wPaper;
    MoveL Offs(pOrigin,222.59,327.15,6.00),vTravel,z5,tPen\WObj:=wPaper;
    MoveL Offs(pOrigin,222.59,327.15,0.00),v60,z0,tPen\WObj:=wPaper;
    MoveL Offs(pOrigin,222.80,326.73,0.00),v40,z0,tPen\WObj:=wPaper;
    MoveL Offs(pOrigin,222.59,327.15,0.00),v40,z0,tPen\WObj:=wPaper;
    MoveL Offs(pOrigin,221.95,327.79,0.00),v40,z0,tPen\WObj:=wPaper;
    MoveL Offs(pOrigin,222.16,327.36,0.00),v40,z0,tPen\WObj:=wPaper;
    MoveL Offs(pOrigin,221.95,327.79,0.00),v40,z0,tPen\WObj:=wPaper;
    MoveL Offs(pOrigin,222.48,328.84,0.00),v40,z0,tPen\WObj:=wPaper;
    MoveL Offs(pOrigin,215.41,335.90,0.00),v40,z0,tPen\WObj:=wPaper;
    MoveL Offs(pOrigin,214.94,334.97,0.00),v40,z0,tPen\WObj:=wPaper;
    MoveL Offs(pOrigin,224.71,334.97,0.00),v40,z0,tPen\WObj:=wPaper;
    MoveL Offs(pOrigin,224.50,334.80,0.00),v40,z0,tPen\WObj:=wPaper;
    MoveL Offs(pOrigin,224.50,335.44,0.00),v40,z0,tPen\WObj:=wPaper;
    MoveL Offs(pOrigin,224.93,335.86,0.00),v40,z0,tPen\WObj:=wPaper;
    MoveL Offs(pOrigin,225.99,336.08,0.00),v40,z0,tPen\WObj:=wPaper;
    MoveL Offs(pOrigin,225.99,336.08,0.00),v40,z0,tPen\WObj:=wPaper;
    MoveL Offs(pOrigin,226.84,335.65,0.00),v40,z0,tPen\WObj:=wPaper;
    MoveL Offs(pOrigin,229.18,335.65,0.00),v40,z0,tPen\WObj:=wPaper;
    MoveL Offs(pOrigin,229.81,334.97,0.00),v40,z0,tPen\WObj:=wPaper;
    MoveL Offs(pOrigin,236.61,334.97,0.00),v40,z0,tPen\WObj:=wPaper;
    MoveL Offs(pOrigin,236.62,335.48,0.00),v40,z0,tPen\WObj:=wPaper;
    MoveL Offs(pOrigin,234.37,333.23,0.00),v40,z0,tPen\WObj:=wPaper;
    MoveL Offs(pOrigin,235.27,332.63,0.00),v40,z0,tPen\WObj:=wPaper;
    MoveL Offs(pOrigin,237.52,334.88,0.00),v40,z0,tPen\WObj:=wPaper;
    MoveL Offs(pOrigin,238.27,334.14,0.00),v40,z0,tPen\WObj:=wPaper;
    MoveL Offs(pOrigin,236.16,332.03,0.00),v40,z0,tPen\WObj:=wPaper;
    MoveL Offs(pOrigin,236.61,333.10,0.00),v40,z0,tPen\WObj:=wPaper;
    MoveL Offs(pOrigin,235.34,334.02,0.00),v40,z0,tPen\WObj:=wPaper;
    MoveL Offs(pOrigin,232.79,335.01,0.00),v40,z0,tPen\WObj:=wPaper;
    MoveL Offs(pOrigin,232.43,334.27,0.00),v40,z0,tPen\WObj:=wPaper;
    MoveL Offs(pOrigin,234.38,336.22,0.00),v40,z0,tPen\WObj:=wPaper;
    MoveL Offs(pOrigin,234.29,336.44,0.00),v40,z0,tPen\WObj:=wPaper;
    MoveL Offs(pOrigin,241.65,329.08,0.00),v40,fine,tPen\WObj:=wPaper;
    MoveL Offs(pOrigin,241.65,329.08,6.00),v60,z5,tPen\WObj:=wPaper;
    MoveL Offs(pOrigin,240.44,326.52,6.00),vTravel,z5,tPen\WObj:=wPaper;
    MoveL Offs(pOrigin,240.44,326.52,0.00),v60,z0,tPen\WObj:=wPaper;
    MoveL Offs(pOrigin,239.38,326.52,0.00),v40,fine,tPen\WObj:=wPaper;
    MoveL Offs(pOrigin,239.38,326.52,6.00),v60,z5,tPen\WObj:=wPaper;
    MoveL Offs(pOrigin,238.67,325.02,6.00),vTravel,z5,tPen\WObj:=wPaper;
    MoveL Offs(pOrigin,238.67,325.02,0.00),v60,z0,tPen\WObj:=wPaper;
    MoveL Offs(pOrigin,238.67,323.54,0.00),v40,fine,tPen\WObj:=wPaper;
    MoveL Offs(pOrigin,238.67,323.54,6.00),v60,z5,tPen\WObj:=wPaper;
    MoveL Offs(pOrigin,242.14,324.60,6.00),vTravel,z5,tPen\WObj:=wPaper;
    MoveL Offs(pOrigin,242.14,324.60,0.00),v60,z0,tPen\WObj:=wPaper;
    MoveL Offs(pOrigin,242.56,325.24,0.00),v40,z0,tPen\WObj:=wPaper;
    MoveL Offs(pOrigin,242.14,324.60,0.00),v40,z0,tPen\WObj:=wPaper;
    MoveL Offs(pOrigin,242.11,325.63,0.00),v40,z0,tPen\WObj:=wPaper;
    MoveL Offs(pOrigin,257.14,310.61,0.00),v40,z0,tPen\WObj:=wPaper;
    MoveL Offs(pOrigin,256.59,310.79,0.00),v40,z0,tPen\WObj:=wPaper;
    MoveL Offs(pOrigin,257.01,311.42,0.00),v40,z0,tPen\WObj:=wPaper;
    MoveL Offs(pOrigin,256.59,310.79,0.00),v40,fine,tPen\WObj:=wPaper;
    MoveL Offs(pOrigin,256.59,310.79,6.00),v60,z5,tPen\WObj:=wPaper;
  ENDPROC

  PROC DrawPart235()
    MoveL Offs(pOrigin,256.47,312.02,6.00),vTravel,z5,tPen\WObj:=wPaper;
    MoveL Offs(pOrigin,256.47,312.02,0.00),v60,z0,tPen\WObj:=wPaper;
    MoveL Offs(pOrigin,274.36,329.90,0.00),v40,z0,tPen\WObj:=wPaper;
    MoveL Offs(pOrigin,274.44,329.06,0.00),v40,z0,tPen\WObj:=wPaper;
    MoveL Offs(pOrigin,275.29,328.21,0.00),v40,z0,tPen\WObj:=wPaper;
    MoveL Offs(pOrigin,275.50,328.85,0.00),v40,z0,tPen\WObj:=wPaper;
    MoveL Offs(pOrigin,275.08,328.63,0.00),v40,z0,tPen\WObj:=wPaper;
    MoveL Offs(pOrigin,271.89,328.63,0.00),v40,z0,tPen\WObj:=wPaper;
    MoveL Offs(pOrigin,270.83,328.42,0.00),v40,z0,tPen\WObj:=wPaper;
    MoveL Offs(pOrigin,270.19,327.58,0.00),v40,z0,tPen\WObj:=wPaper;
    MoveL Offs(pOrigin,269.98,326.09,0.00),v40,z0,tPen\WObj:=wPaper;
    MoveL Offs(pOrigin,269.98,326.09,0.00),v40,z0,tPen\WObj:=wPaper;
    MoveL Offs(pOrigin,269.41,324.60,0.00),v40,z0,tPen\WObj:=wPaper;
    MoveL Offs(pOrigin,267.00,320.99,0.00),v40,z0,tPen\WObj:=wPaper;
    MoveL Offs(pOrigin,267.00,320.99,0.00),v40,z0,tPen\WObj:=wPaper;
    MoveL Offs(pOrigin,263.81,319.50,0.00),v40,fine,tPen\WObj:=wPaper;
    MoveL Offs(pOrigin,263.81,319.50,6.00),v60,z5,tPen\WObj:=wPaper;
    MoveL Offs(pOrigin,264.45,321.41,6.00),vTravel,z5,tPen\WObj:=wPaper;
    MoveL Offs(pOrigin,264.45,321.41,0.00),v60,z0,tPen\WObj:=wPaper;
    MoveL Offs(pOrigin,262.33,320.00,0.00),v40,z0,tPen\WObj:=wPaper;
    MoveL Offs(pOrigin,261.26,319.71,0.00),v40,z0,tPen\WObj:=wPaper;
    MoveL Offs(pOrigin,261.48,319.13,0.00),v40,z0,tPen\WObj:=wPaper;
    MoveL Offs(pOrigin,266.79,319.13,0.00),v40,fine,tPen\WObj:=wPaper;
    MoveL Offs(pOrigin,266.79,319.13,6.00),v60,z5,tPen\WObj:=wPaper;
    MoveL Offs(pOrigin,266.58,320.77,6.00),vTravel,z5,tPen\WObj:=wPaper;
    MoveL Offs(pOrigin,266.58,320.77,0.00),v60,z0,tPen\WObj:=wPaper;
    MoveL Offs(pOrigin,267.00,320.99,0.00),v40,z0,tPen\WObj:=wPaper;
    MoveL Offs(pOrigin,266.58,320.77,0.00),v40,z0,tPen\WObj:=wPaper;
    MoveL Offs(pOrigin,265.73,321.24,0.00),v40,z0,tPen\WObj:=wPaper;
    MoveL Offs(pOrigin,259.14,321.24,0.00),v40,z0,tPen\WObj:=wPaper;
    MoveL Offs(pOrigin,258.71,321.20,0.00),v40,z0,tPen\WObj:=wPaper;
    MoveL Offs(pOrigin,259.35,321.84,0.00),v40,z0,tPen\WObj:=wPaper;
    MoveL Offs(pOrigin,258.71,321.20,0.00),v40,z0,tPen\WObj:=wPaper;
    MoveL Offs(pOrigin,258.73,320.77,0.00),v40,z0,tPen\WObj:=wPaper;
    MoveL Offs(pOrigin,258.73,319.29,0.00),v40,z0,tPen\WObj:=wPaper;
    MoveL Offs(pOrigin,257.68,318.86,0.00),v40,z0,tPen\WObj:=wPaper;
    MoveL Offs(pOrigin,257.68,320.35,0.00),v40,fine,tPen\WObj:=wPaper;
    MoveL Offs(pOrigin,257.68,320.35,6.00),v60,z5,tPen\WObj:=wPaper;
    MoveL Offs(pOrigin,256.62,319.71,6.00),vTravel,z5,tPen\WObj:=wPaper;
    MoveL Offs(pOrigin,256.62,319.71,0.00),v60,z0,tPen\WObj:=wPaper;
    MoveL Offs(pOrigin,256.62,315.25,0.00),v40,z0,tPen\WObj:=wPaper;
    MoveL Offs(pOrigin,257.68,315.68,0.00),v40,z0,tPen\WObj:=wPaper;
    MoveL Offs(pOrigin,257.68,317.38,0.00),v40,fine,tPen\WObj:=wPaper;
    MoveL Offs(pOrigin,257.68,317.38,6.00),v60,z5,tPen\WObj:=wPaper;
    MoveL Offs(pOrigin,259.79,319.92,6.00),vTravel,z5,tPen\WObj:=wPaper;
    MoveL Offs(pOrigin,259.79,319.92,0.00),v60,z0,tPen\WObj:=wPaper;
    MoveL Offs(pOrigin,259.79,321.41,0.00),v40,z0,tPen\WObj:=wPaper;
    MoveL Offs(pOrigin,259.35,322.37,0.00),v40,z0,tPen\WObj:=wPaper;
    MoveL Offs(pOrigin,250.64,313.65,0.00),v40,z0,tPen\WObj:=wPaper;
    MoveL Offs(pOrigin,251.49,313.85,0.00),v40,z0,tPen\WObj:=wPaper;
    MoveL Offs(pOrigin,255.52,313.85,0.00),v40,z0,tPen\WObj:=wPaper;
    MoveL Offs(pOrigin,255.52,313.55,0.00),v40,z0,tPen\WObj:=wPaper;
    MoveL Offs(pOrigin,255.95,313.98,0.00),v40,z0,tPen\WObj:=wPaper;
    MoveL Offs(pOrigin,255.52,313.55,0.00),v40,z0,tPen\WObj:=wPaper;
    MoveL Offs(pOrigin,255.57,314.61,0.00),v40,z0,tPen\WObj:=wPaper;
    MoveL Offs(pOrigin,255.57,321.41,0.00),v40,z0,tPen\WObj:=wPaper;
    MoveL Offs(pOrigin,255.52,322.26,0.00),v40,z0,tPen\WObj:=wPaper;
    MoveL Offs(pOrigin,254.68,321.20,0.00),v40,z0,tPen\WObj:=wPaper;
    MoveL Offs(pOrigin,252.55,319.85,0.00),v40,z0,tPen\WObj:=wPaper;
    MoveL Offs(pOrigin,252.12,319.08,0.00),v40,z0,tPen\WObj:=wPaper;
    MoveL Offs(pOrigin,252.12,319.08,0.00),v40,z0,tPen\WObj:=wPaper;
    MoveL Offs(pOrigin,252.34,317.16,0.00),v40,fine,tPen\WObj:=wPaper;
    MoveL Offs(pOrigin,252.34,317.16,6.00),v60,z5,tPen\WObj:=wPaper;
    MoveL Offs(pOrigin,251.34,318.01,6.00),vTravel,z5,tPen\WObj:=wPaper;
    MoveL Offs(pOrigin,251.34,318.01,0.00),v60,z0,tPen\WObj:=wPaper;
    MoveL Offs(pOrigin,251.34,320.99,0.00),v40,z0,tPen\WObj:=wPaper;
    MoveL Offs(pOrigin,252.40,320.56,0.00),v40,z0,tPen\WObj:=wPaper;
    MoveL Offs(pOrigin,252.40,321.62,0.00),v40,z0,tPen\WObj:=wPaper;
    MoveL Offs(pOrigin,252.76,322.30,0.00),v40,z0,tPen\WObj:=wPaper;
    MoveL Offs(pOrigin,258.08,322.30,0.00),v40,z0,tPen\WObj:=wPaper;
    MoveL Offs(pOrigin,257.68,322.90,0.00),v40,z0,tPen\WObj:=wPaper;
    MoveL Offs(pOrigin,257.68,324.60,0.00),v40,z0,tPen\WObj:=wPaper;
    MoveL Offs(pOrigin,257.44,324.41,0.00),v40,z0,tPen\WObj:=wPaper;
    MoveL Offs(pOrigin,259.14,324.41,0.00),v40,z0,tPen\WObj:=wPaper;
    MoveL Offs(pOrigin,259.14,324.17,0.00),v40,z0,tPen\WObj:=wPaper;
    MoveL Offs(pOrigin,259.56,324.25,0.00),v40,z0,tPen\WObj:=wPaper;
    MoveL Offs(pOrigin,260.06,325.02,0.00),v40,z0,tPen\WObj:=wPaper;
    MoveL Offs(pOrigin,261.05,328.85,0.00),v40,z0,tPen\WObj:=wPaper;
    MoveL Offs(pOrigin,260.48,331.61,0.00),v40,z0,tPen\WObj:=wPaper;
    MoveL Offs(pOrigin,259.77,332.25,0.00),v40,z0,tPen\WObj:=wPaper;
    MoveL Offs(pOrigin,260.51,332.62,0.00),v40,z0,tPen\WObj:=wPaper;
    MoveL Offs(pOrigin,253.45,339.68,0.00),v40,z0,tPen\WObj:=wPaper;
    MoveL Offs(pOrigin,253.86,339.28,0.00),v40,z0,tPen\WObj:=wPaper;
    MoveL Offs(pOrigin,251.61,337.03,0.00),v40,fine,tPen\WObj:=wPaper;
    MoveL Offs(pOrigin,251.61,337.03,6.00),v60,z5,tPen\WObj:=wPaper;
    MoveL Offs(pOrigin,252.98,335.86,6.00),vTravel,z5,tPen\WObj:=wPaper;
    MoveL Offs(pOrigin,252.98,335.86,0.00),v60,z0,tPen\WObj:=wPaper;
    MoveL Offs(pOrigin,252.62,336.92,0.00),v40,z0,tPen\WObj:=wPaper;
    MoveL Offs(pOrigin,254.04,337.14,0.00),v40,z0,tPen\WObj:=wPaper;
    MoveL Offs(pOrigin,253.45,337.35,0.00),v40,z0,tPen\WObj:=wPaper;
    MoveL Offs(pOrigin,253.45,338.62,0.00),v40,fine,tPen\WObj:=wPaper;
    MoveL Offs(pOrigin,253.45,338.62,6.00),v60,z5,tPen\WObj:=wPaper;
    MoveL Offs(pOrigin,255.10,339.53,6.00),vTravel,z5,tPen\WObj:=wPaper;
    MoveL Offs(pOrigin,255.10,339.53,0.00),v60,z0,tPen\WObj:=wPaper;
    MoveL Offs(pOrigin,264.27,330.36,0.00),v40,fine,tPen\WObj:=wPaper;
    MoveL Offs(pOrigin,264.27,330.36,6.00),v60,z5,tPen\WObj:=wPaper;
    MoveL Offs(pOrigin,265.46,330.66,6.00),vTravel,z5,tPen\WObj:=wPaper;
    MoveL Offs(pOrigin,265.46,330.66,0.00),v60,z0,tPen\WObj:=wPaper;
    MoveL Offs(pOrigin,273.13,322.99,0.00),v40,z0,tPen\WObj:=wPaper;
    MoveL Offs(pOrigin,272.74,323.54,0.00),v40,z0,tPen\WObj:=wPaper;
    MoveL Offs(pOrigin,274.01,323.54,0.00),v40,z0,tPen\WObj:=wPaper;
    MoveL Offs(pOrigin,277.62,324.39,0.00),v40,z0,tPen\WObj:=wPaper;
    MoveL Offs(pOrigin,281.66,323.11,0.00),v40,z0,tPen\WObj:=wPaper;
    MoveL Offs(pOrigin,281.45,322.55,0.00),v40,z0,tPen\WObj:=wPaper;
    MoveL Offs(pOrigin,279.75,322.26,0.00),v40,z0,tPen\WObj:=wPaper;
    MoveL Offs(pOrigin,279.75,321.62,0.00),v40,z0,tPen\WObj:=wPaper;
    MoveL Offs(pOrigin,278.26,320.99,0.00),v40,z0,tPen\WObj:=wPaper;
    MoveL Offs(pOrigin,277.41,320.99,0.00),v40,z0,tPen\WObj:=wPaper;
    MoveL Offs(pOrigin,277.33,320.28,0.00),v40,z0,tPen\WObj:=wPaper;
    MoveL Offs(pOrigin,276.43,321.19,0.00),v40,z0,tPen\WObj:=wPaper;
    MoveL Offs(pOrigin,277.32,321.78,0.00),v40,z0,tPen\WObj:=wPaper;
    MoveL Offs(pOrigin,278.38,320.73,0.00),v40,z0,tPen\WObj:=wPaper;
    MoveL Offs(pOrigin,279.42,321.18,0.00),v40,z0,tPen\WObj:=wPaper;
    MoveL Offs(pOrigin,278.37,322.23,0.00),v40,fine,tPen\WObj:=wPaper;
    MoveL Offs(pOrigin,278.37,322.23,6.00),v60,z5,tPen\WObj:=wPaper;
    MoveL Offs(pOrigin,277.78,324.37,6.00),vTravel,z5,tPen\WObj:=wPaper;
    MoveL Offs(pOrigin,277.78,324.37,0.00),v60,z0,tPen\WObj:=wPaper;
    MoveL Offs(pOrigin,280.34,326.93,0.00),v40,z0,tPen\WObj:=wPaper;
    MoveL Offs(pOrigin,280.45,327.61,0.00),v40,z0,tPen\WObj:=wPaper;
    MoveL Offs(pOrigin,290.37,317.70,0.00),v40,z0,tPen\WObj:=wPaper;
  ENDPROC

  PROC DrawPart236()
    MoveL Offs(pOrigin,290.05,317.22,0.00),v40,z0,tPen\WObj:=wPaper;
    MoveL Offs(pOrigin,287.79,314.97,0.00),v40,z0,tPen\WObj:=wPaper;
    MoveL Offs(pOrigin,288.46,315.04,0.00),v40,z0,tPen\WObj:=wPaper;
    MoveL Offs(pOrigin,287.19,315.11,0.00),v40,z0,tPen\WObj:=wPaper;
    MoveL Offs(pOrigin,286.62,315.89,0.00),v40,z0,tPen\WObj:=wPaper;
    MoveL Offs(pOrigin,286.98,316.10,0.00),v40,z0,tPen\WObj:=wPaper;
    MoveL Offs(pOrigin,288.46,315.46,0.00),v40,z0,tPen\WObj:=wPaper;
    MoveL Offs(pOrigin,288.46,315.46,0.00),v40,z0,tPen\WObj:=wPaper;
    MoveL Offs(pOrigin,288.18,316.74,0.00),v40,z0,tPen\WObj:=wPaper;
    MoveL Offs(pOrigin,287.19,317.80,0.00),v40,z0,tPen\WObj:=wPaper;
    MoveL Offs(pOrigin,286.98,318.07,0.00),v40,z0,tPen\WObj:=wPaper;
    MoveL Offs(pOrigin,289.10,318.07,0.00),v40,z0,tPen\WObj:=wPaper;
    MoveL Offs(pOrigin,289.60,318.27,0.00),v40,z0,tPen\WObj:=wPaper;
    MoveL Offs(pOrigin,287.35,316.01,0.00),v40,z0,tPen\WObj:=wPaper;
    MoveL Offs(pOrigin,286.55,316.10,0.00),v40,z0,tPen\WObj:=wPaper;
    MoveL Offs(pOrigin,284.42,317.30,0.00),v40,z0,tPen\WObj:=wPaper;
    MoveL Offs(pOrigin,283.36,317.38,0.00),v40,z0,tPen\WObj:=wPaper;
    MoveL Offs(pOrigin,283.03,317.57,0.00),v40,z0,tPen\WObj:=wPaper;
    MoveL Offs(pOrigin,284.38,316.22,0.00),v40,z0,tPen\WObj:=wPaper;
    MoveL Offs(pOrigin,284.85,316.74,0.00),v40,z0,tPen\WObj:=wPaper;
    MoveL Offs(pOrigin,283.36,316.52,0.00),v40,z0,tPen\WObj:=wPaper;
    MoveL Offs(pOrigin,282.88,316.22,0.00),v40,z0,tPen\WObj:=wPaper;
    MoveL Offs(pOrigin,281.68,317.42,0.00),v40,z0,tPen\WObj:=wPaper;
    MoveL Offs(pOrigin,280.64,316.98,0.00),v40,z0,tPen\WObj:=wPaper;
    MoveL Offs(pOrigin,281.54,316.08,0.00),v40,fine,tPen\WObj:=wPaper;
    MoveL Offs(pOrigin,281.54,316.08,6.00),v60,z5,tPen\WObj:=wPaper;
    MoveL Offs(pOrigin,281.54,314.58,6.00),vTravel,z5,tPen\WObj:=wPaper;
    MoveL Offs(pOrigin,281.54,314.58,0.00),v60,z0,tPen\WObj:=wPaper;
    MoveL Offs(pOrigin,298.07,298.05,0.00),v40,fine,tPen\WObj:=wPaper;
    MoveL Offs(pOrigin,298.07,298.05,6.00),v60,z5,tPen\WObj:=wPaper;
    MoveL Offs(pOrigin,297.18,296.95,6.00),vTravel,z5,tPen\WObj:=wPaper;
    MoveL Offs(pOrigin,297.18,296.95,0.00),v60,z0,tPen\WObj:=wPaper;
    MoveL Offs(pOrigin,293.99,296.95,0.00),v40,fine,tPen\WObj:=wPaper;
    MoveL Offs(pOrigin,293.99,296.95,6.00),v60,z5,tPen\WObj:=wPaper;
    MoveL Offs(pOrigin,293.58,298.46,6.00),vTravel,z5,tPen\WObj:=wPaper;
    MoveL Offs(pOrigin,293.58,298.46,0.00),v60,z0,tPen\WObj:=wPaper;
    MoveL Offs(pOrigin,293.58,299.95,0.00),v40,z0,tPen\WObj:=wPaper;
    MoveL Offs(pOrigin,292.53,299.95,0.00),v40,z0,tPen\WObj:=wPaper;
    MoveL Offs(pOrigin,292.53,298.89,0.00),v40,fine,tPen\WObj:=wPaper;
    MoveL Offs(pOrigin,292.53,298.89,6.00),v60,z5,tPen\WObj:=wPaper;
    MoveL Offs(pOrigin,294.64,298.68,6.00),vTravel,z5,tPen\WObj:=wPaper;
    MoveL Offs(pOrigin,294.64,298.68,0.00),v60,z0,tPen\WObj:=wPaper;
    MoveL Offs(pOrigin,294.64,300.16,0.00),v40,fine,tPen\WObj:=wPaper;
    MoveL Offs(pOrigin,294.64,300.16,6.00),v60,z5,tPen\WObj:=wPaper;
    MoveL Offs(pOrigin,296.32,302.23,6.00),vTravel,z5,tPen\WObj:=wPaper;
    MoveL Offs(pOrigin,296.32,302.23,0.00),v60,z0,tPen\WObj:=wPaper;
    MoveL Offs(pOrigin,292.50,302.23,0.00),v40,fine,tPen\WObj:=wPaper;
    MoveL Offs(pOrigin,292.50,302.23,6.00),v60,z5,tPen\WObj:=wPaper;
    MoveL Offs(pOrigin,290.80,302.23,6.00),vTravel,z5,tPen\WObj:=wPaper;
    MoveL Offs(pOrigin,290.80,302.23,0.00),v60,z0,tPen\WObj:=wPaper;
    MoveL Offs(pOrigin,288.46,302.23,0.00),v40,z0,tPen\WObj:=wPaper;
    MoveL Offs(pOrigin,289.36,301.86,0.00),v40,z0,tPen\WObj:=wPaper;
    MoveL Offs(pOrigin,289.36,302.92,0.00),v40,fine,tPen\WObj:=wPaper;
    MoveL Offs(pOrigin,289.36,302.92,6.00),v60,z5,tPen\WObj:=wPaper;
    MoveL Offs(pOrigin,289.31,304.34,6.00),vTravel,z5,tPen\WObj:=wPaper;
    MoveL Offs(pOrigin,289.31,304.34,0.00),v60,z0,tPen\WObj:=wPaper;
    MoveL Offs(pOrigin,288.04,304.34,0.00),v40,z0,tPen\WObj:=wPaper;
    MoveL Offs(pOrigin,287.31,304.03,0.00),v40,z0,tPen\WObj:=wPaper;
    MoveL Offs(pOrigin,293.47,310.19,0.00),v40,z0,tPen\WObj:=wPaper;
    MoveL Offs(pOrigin,293.83,311.24,0.00),v40,z0,tPen\WObj:=wPaper;
    MoveL Offs(pOrigin,275.80,329.28,0.00),v40,z0,tPen\WObj:=wPaper;
    MoveL Offs(pOrigin,275.10,329.16,0.00),v40,z0,tPen\WObj:=wPaper;
    MoveL Offs(pOrigin,271.50,325.55,0.00),v40,z0,tPen\WObj:=wPaper;
    MoveL Offs(pOrigin,271.46,326.52,0.00),v40,z0,tPen\WObj:=wPaper;
    MoveL Offs(pOrigin,273.80,326.52,0.00),v40,z0,tPen\WObj:=wPaper;
    MoveL Offs(pOrigin,273.90,326.46,0.00),v40,z0,tPen\WObj:=wPaper;
    MoveL Offs(pOrigin,276.00,328.56,0.00),v40,fine,tPen\WObj:=wPaper;
    MoveL Offs(pOrigin,276.00,328.56,6.00),v60,z5,tPen\WObj:=wPaper;
    MoveL Offs(pOrigin,274.57,328.42,6.00),vTravel,z5,tPen\WObj:=wPaper;
    MoveL Offs(pOrigin,274.57,328.42,0.00),v60,z0,tPen\WObj:=wPaper;
    MoveL Offs(pOrigin,274.57,327.36,0.00),v40,z0,tPen\WObj:=wPaper;
    MoveL Offs(pOrigin,273.52,327.36,0.00),v40,z0,tPen\WObj:=wPaper;
    MoveL Offs(pOrigin,273.52,328.64,0.00),v40,z0,tPen\WObj:=wPaper;
    MoveL Offs(pOrigin,273.16,328.85,0.00),v40,z0,tPen\WObj:=wPaper;
    MoveL Offs(pOrigin,273.16,327.79,0.00),v40,z0,tPen\WObj:=wPaper;
    MoveL Offs(pOrigin,273.16,327.79,0.00),v40,z0,tPen\WObj:=wPaper;
    MoveL Offs(pOrigin,271.46,327.15,0.00),v40,z0,tPen\WObj:=wPaper;
    MoveL Offs(pOrigin,271.46,327.15,0.00),v40,z0,tPen\WObj:=wPaper;
    MoveL Offs(pOrigin,270.61,326.09,0.00),v40,z0,tPen\WObj:=wPaper;
    MoveL Offs(pOrigin,270.61,326.09,0.00),v40,z0,tPen\WObj:=wPaper;
    MoveL Offs(pOrigin,271.25,325.45,0.00),v40,z0,tPen\WObj:=wPaper;
    MoveL Offs(pOrigin,275.29,326.73,0.00),v40,z0,tPen\WObj:=wPaper;
    MoveL Offs(pOrigin,277.62,326.73,0.00),v40,z0,tPen\WObj:=wPaper;
    MoveL Offs(pOrigin,279.75,326.09,0.00),v40,fine,tPen\WObj:=wPaper;
    MoveL Offs(pOrigin,279.75,326.09,6.00),v60,z5,tPen\WObj:=wPaper;
    MoveL Offs(pOrigin,278.09,327.67,6.00),vTravel,z5,tPen\WObj:=wPaper;
    MoveL Offs(pOrigin,278.09,327.67,0.00),v60,z0,tPen\WObj:=wPaper;
    MoveL Offs(pOrigin,276.89,326.47,0.00),v40,fine,tPen\WObj:=wPaper;
    MoveL Offs(pOrigin,276.89,326.47,6.00),v60,z5,tPen\WObj:=wPaper;
    MoveL Offs(pOrigin,274.44,329.06,6.00),vTravel,z5,tPen\WObj:=wPaper;
    MoveL Offs(pOrigin,274.44,329.06,0.00),v60,z0,tPen\WObj:=wPaper;
    MoveL Offs(pOrigin,273.16,328.85,0.00),v40,fine,tPen\WObj:=wPaper;
    MoveL Offs(pOrigin,273.16,328.85,6.00),v60,z5,tPen\WObj:=wPaper;
    MoveL Offs(pOrigin,273.46,330.50,6.00),vTravel,z5,tPen\WObj:=wPaper;
    MoveL Offs(pOrigin,273.46,330.50,0.00),v60,z0,tPen\WObj:=wPaper;
    MoveL Offs(pOrigin,256.63,313.67,0.00),v40,fine,tPen\WObj:=wPaper;
    MoveL Offs(pOrigin,256.63,313.67,6.00),v60,z5,tPen\WObj:=wPaper;
    MoveL Offs(pOrigin,258.29,312.27,6.00),vTravel,z5,tPen\WObj:=wPaper;
    MoveL Offs(pOrigin,258.29,312.27,0.00),v60,z0,tPen\WObj:=wPaper;
    MoveL Offs(pOrigin,258.71,312.70,0.00),v40,z0,tPen\WObj:=wPaper;
    MoveL Offs(pOrigin,258.29,312.27,0.00),v40,fine,tPen\WObj:=wPaper;
    MoveL Offs(pOrigin,258.29,312.27,6.00),v60,z5,tPen\WObj:=wPaper;
    MoveL Offs(pOrigin,262.02,311.59,6.00),vTravel,z5,tPen\WObj:=wPaper;
    MoveL Offs(pOrigin,262.02,311.59,0.00),v60,z0,tPen\WObj:=wPaper;
    MoveL Offs(pOrigin,269.53,319.10,0.00),v40,fine,tPen\WObj:=wPaper;
    MoveL Offs(pOrigin,269.53,319.10,6.00),v60,z5,tPen\WObj:=wPaper;
    MoveL Offs(pOrigin,270.59,321.05,6.00),vTravel,z5,tPen\WObj:=wPaper;
    MoveL Offs(pOrigin,270.59,321.05,0.00),v60,z0,tPen\WObj:=wPaper;
    MoveL Offs(pOrigin,265.18,326.46,0.00),v40,z0,tPen\WObj:=wPaper;
    MoveL Offs(pOrigin,266.36,326.52,0.00),v40,z0,tPen\WObj:=wPaper;
    MoveL Offs(pOrigin,268.49,326.52,0.00),v40,z0,tPen\WObj:=wPaper;
    MoveL Offs(pOrigin,268.27,326.73,0.00),v40,z0,tPen\WObj:=wPaper;
    MoveL Offs(pOrigin,269.55,326.51,0.00),v40,z0,tPen\WObj:=wPaper;
    MoveL Offs(pOrigin,269.98,326.09,0.00),v40,z0,tPen\WObj:=wPaper;
    MoveL Offs(pOrigin,270.19,326.09,0.00),v40,z0,tPen\WObj:=wPaper;
    MoveL Offs(pOrigin,271.04,326.73,0.00),v40,fine,tPen\WObj:=wPaper;
    MoveL Offs(pOrigin,271.04,326.73,6.00),v60,z5,tPen\WObj:=wPaper;
    MoveL Offs(pOrigin,270.40,328.42,6.00),vTravel,z5,tPen\WObj:=wPaper;
    MoveL Offs(pOrigin,270.40,328.42,0.00),v60,z0,tPen\WObj:=wPaper;
    MoveL Offs(pOrigin,270.83,330.27,0.00),v40,z0,tPen\WObj:=wPaper;
  ENDPROC

  PROC DrawPart237()
    MoveL Offs(pOrigin,269.12,330.27,0.00),v40,z0,tPen\WObj:=wPaper;
    MoveL Offs(pOrigin,268.91,328.42,0.00),v40,z0,tPen\WObj:=wPaper;
    MoveL Offs(pOrigin,268.27,327.58,0.00),v40,z0,tPen\WObj:=wPaper;
    MoveL Offs(pOrigin,268.49,327.58,0.00),v40,z0,tPen\WObj:=wPaper;
    MoveL Offs(pOrigin,266.58,327.58,0.00),v40,fine,tPen\WObj:=wPaper;
    MoveL Offs(pOrigin,266.58,327.58,6.00),v60,z5,tPen\WObj:=wPaper;
    MoveL Offs(pOrigin,267.18,325.88,6.00),vTravel,z5,tPen\WObj:=wPaper;
    MoveL Offs(pOrigin,267.18,325.88,0.00),v60,z0,tPen\WObj:=wPaper;
    MoveL Offs(pOrigin,267.18,329.49,0.00),v40,fine,tPen\WObj:=wPaper;
    MoveL Offs(pOrigin,267.18,329.49,6.00),v60,z5,tPen\WObj:=wPaper;
    MoveL Offs(pOrigin,264.42,328.71,6.00),vTravel,z5,tPen\WObj:=wPaper;
    MoveL Offs(pOrigin,264.42,328.71,0.00),v60,z0,tPen\WObj:=wPaper;
    MoveL Offs(pOrigin,262.77,330.36,0.00),v40,fine,tPen\WObj:=wPaper;
    MoveL Offs(pOrigin,262.77,330.36,6.00),v60,z5,tPen\WObj:=wPaper;
    MoveL Offs(pOrigin,262.96,331.61,6.00),vTravel,z5,tPen\WObj:=wPaper;
    MoveL Offs(pOrigin,262.96,331.61,0.00),v60,z0,tPen\WObj:=wPaper;
    MoveL Offs(pOrigin,263.39,328.85,0.00),v40,z0,tPen\WObj:=wPaper;
    MoveL Offs(pOrigin,262.61,325.88,0.00),v40,z0,tPen\WObj:=wPaper;
    MoveL Offs(pOrigin,260.20,322.69,0.00),v40,z0,tPen\WObj:=wPaper;
    MoveL Offs(pOrigin,258.50,321.27,0.00),v40,z0,tPen\WObj:=wPaper;
    MoveL Offs(pOrigin,257.86,321.13,0.00),v40,z0,tPen\WObj:=wPaper;
    MoveL Offs(pOrigin,257.72,321.62,0.00),v40,z0,tPen\WObj:=wPaper;
    MoveL Offs(pOrigin,259.07,323.33,0.00),v40,z0,tPen\WObj:=wPaper;
    MoveL Offs(pOrigin,259.14,324.17,0.00),v40,z0,tPen\WObj:=wPaper;
    MoveL Offs(pOrigin,259.14,324.17,0.00),v40,z0,tPen\WObj:=wPaper;
    MoveL Offs(pOrigin,258.71,324.81,0.00),v40,z0,tPen\WObj:=wPaper;
    MoveL Offs(pOrigin,259.77,328.00,0.00),v40,z0,tPen\WObj:=wPaper;
    MoveL Offs(pOrigin,259.77,329.70,0.00),v40,z0,tPen\WObj:=wPaper;
    MoveL Offs(pOrigin,259.35,331.40,0.00),v40,z0,tPen\WObj:=wPaper;
    MoveL Offs(pOrigin,259.77,333.10,0.00),v40,z0,tPen\WObj:=wPaper;
    MoveL Offs(pOrigin,258.43,335.01,0.00),v40,z0,tPen\WObj:=wPaper;
    MoveL Offs(pOrigin,257.65,335.44,0.00),v40,z0,tPen\WObj:=wPaper;
    MoveL Offs(pOrigin,257.86,334.97,0.00),v40,z0,tPen\WObj:=wPaper;
    MoveL Offs(pOrigin,255.31,334.97,0.00),v40,z0,tPen\WObj:=wPaper;
    MoveL Offs(pOrigin,255.20,334.64,0.00),v40,z0,tPen\WObj:=wPaper;
    MoveL Offs(pOrigin,258.35,337.80,0.00),v40,z0,tPen\WObj:=wPaper;
    MoveL Offs(pOrigin,257.30,338.24,0.00),v40,z0,tPen\WObj:=wPaper;
    MoveL Offs(pOrigin,254.30,335.24,0.00),v40,fine,tPen\WObj:=wPaper;
    MoveL Offs(pOrigin,254.30,335.24,6.00),v60,z5,tPen\WObj:=wPaper;
    MoveL Offs(pOrigin,252.34,334.80,6.00),vTravel,z5,tPen\WObj:=wPaper;
    MoveL Offs(pOrigin,252.34,334.80,0.00),v60,z0,tPen\WObj:=wPaper;
    MoveL Offs(pOrigin,254.60,332.46,0.00),v40,z0,tPen\WObj:=wPaper;
    MoveL Offs(pOrigin,255.31,330.76,0.00),v40,fine,tPen\WObj:=wPaper;
    MoveL Offs(pOrigin,255.31,330.76,6.00),v60,z5,tPen\WObj:=wPaper;
    MoveL Offs(pOrigin,257.53,329.63,6.00),vTravel,z5,tPen\WObj:=wPaper;
    MoveL Offs(pOrigin,257.53,329.63,0.00),v60,z0,tPen\WObj:=wPaper;
    MoveL Offs(pOrigin,260.68,326.48,0.00),v40,fine,tPen\WObj:=wPaper;
    MoveL Offs(pOrigin,260.68,326.48,6.00),v60,z5,tPen\WObj:=wPaper;
    MoveL Offs(pOrigin,259.35,325.46,6.00),vTravel,z5,tPen\WObj:=wPaper;
    MoveL Offs(pOrigin,259.35,325.46,0.00),v60,z0,tPen\WObj:=wPaper;
    MoveL Offs(pOrigin,258.08,325.46,0.00),v40,fine,tPen\WObj:=wPaper;
    MoveL Offs(pOrigin,258.08,325.46,6.00),v60,z5,tPen\WObj:=wPaper;
    MoveL Offs(pOrigin,257.23,324.39,6.00),vTravel,z5,tPen\WObj:=wPaper;
    MoveL Offs(pOrigin,257.23,324.39,0.00),v60,z0,tPen\WObj:=wPaper;
    MoveL Offs(pOrigin,257.44,324.81,0.00),v40,z0,tPen\WObj:=wPaper;
    MoveL Offs(pOrigin,257.23,324.39,0.00),v40,z0,tPen\WObj:=wPaper;
    MoveL Offs(pOrigin,256.16,324.17,0.00),v40,z0,tPen\WObj:=wPaper;
    MoveL Offs(pOrigin,255.60,322.48,0.00),v40,z0,tPen\WObj:=wPaper;
    MoveL Offs(pOrigin,256.80,322.69,0.00),v40,z0,tPen\WObj:=wPaper;
    MoveL Offs(pOrigin,256.62,323.32,0.00),v40,z0,tPen\WObj:=wPaper;
    MoveL Offs(pOrigin,256.62,321.62,0.00),v40,fine,tPen\WObj:=wPaper;
    MoveL Offs(pOrigin,256.62,321.62,6.00),v60,z5,tPen\WObj:=wPaper;
    MoveL Offs(pOrigin,255.95,323.75,6.00),vTravel,z5,tPen\WObj:=wPaper;
    MoveL Offs(pOrigin,255.95,323.75,0.00),v60,z0,tPen\WObj:=wPaper;
    MoveL Offs(pOrigin,256.16,324.17,0.00),v40,z0,tPen\WObj:=wPaper;
    MoveL Offs(pOrigin,255.95,323.75,0.00),v40,fine,tPen\WObj:=wPaper;
    MoveL Offs(pOrigin,255.95,323.75,6.00),v60,z5,tPen\WObj:=wPaper;
    MoveL Offs(pOrigin,253.45,322.47,6.00),vTravel,z5,tPen\WObj:=wPaper;
    MoveL Offs(pOrigin,253.45,322.47,0.00),v60,z0,tPen\WObj:=wPaper;
    MoveL Offs(pOrigin,253.45,321.20,0.00),v40,fine,tPen\WObj:=wPaper;
    MoveL Offs(pOrigin,253.45,321.20,6.00),v60,z5,tPen\WObj:=wPaper;
    MoveL Offs(pOrigin,254.51,320.56,6.00),vTravel,z5,tPen\WObj:=wPaper;
    MoveL Offs(pOrigin,254.51,320.56,0.00),v60,z0,tPen\WObj:=wPaper;
    MoveL Offs(pOrigin,254.51,316.31,0.00),v40,fine,tPen\WObj:=wPaper;
    MoveL Offs(pOrigin,254.51,316.31,6.00),v60,z5,tPen\WObj:=wPaper;
    MoveL Offs(pOrigin,253.45,315.04,6.00),vTravel,z5,tPen\WObj:=wPaper;
    MoveL Offs(pOrigin,253.45,315.04,0.00),v60,z0,tPen\WObj:=wPaper;
    MoveL Offs(pOrigin,253.45,319.71,0.00),v40,z0,tPen\WObj:=wPaper;
    MoveL Offs(pOrigin,252.40,319.29,0.00),v40,z0,tPen\WObj:=wPaper;
    MoveL Offs(pOrigin,252.40,314.19,0.00),v40,z0,tPen\WObj:=wPaper;
    MoveL Offs(pOrigin,253.19,313.98,0.00),v40,z0,tPen\WObj:=wPaper;
    MoveL Offs(pOrigin,253.82,314.61,0.00),v40,z0,tPen\WObj:=wPaper;
    MoveL Offs(pOrigin,253.19,313.98,0.00),v40,fine,tPen\WObj:=wPaper;
    MoveL Offs(pOrigin,253.19,313.98,6.00),v60,z5,tPen\WObj:=wPaper;
    MoveL Offs(pOrigin,253.78,312.32,6.00),vTravel,z5,tPen\WObj:=wPaper;
    MoveL Offs(pOrigin,253.78,312.32,0.00),v60,z0,tPen\WObj:=wPaper;
    MoveL Offs(pOrigin,272.56,331.10,0.00),v40,z0,tPen\WObj:=wPaper;
    MoveL Offs(pOrigin,272.52,331.61,0.00),v40,z0,tPen\WObj:=wPaper;
    MoveL Offs(pOrigin,272.10,332.04,0.00),v40,z0,tPen\WObj:=wPaper;
    MoveL Offs(pOrigin,272.52,331.61,0.00),v40,fine,tPen\WObj:=wPaper;
    MoveL Offs(pOrigin,272.52,331.61,6.00),v60,z5,tPen\WObj:=wPaper;
    MoveL Offs(pOrigin,273.59,330.55,6.00),vTravel,z5,tPen\WObj:=wPaper;
    MoveL Offs(pOrigin,273.59,330.55,0.00),v60,z0,tPen\WObj:=wPaper;
    MoveL Offs(pOrigin,272.95,331.19,0.00),v40,z0,tPen\WObj:=wPaper;
    MoveL Offs(pOrigin,273.59,330.55,0.00),v40,fine,tPen\WObj:=wPaper;
    MoveL Offs(pOrigin,273.59,330.55,6.00),v60,z5,tPen\WObj:=wPaper;
    MoveL Offs(pOrigin,269.12,325.46,6.00),vTravel,z5,tPen\WObj:=wPaper;
    MoveL Offs(pOrigin,269.12,325.46,0.00),v60,z0,tPen\WObj:=wPaper;
    MoveL Offs(pOrigin,265.94,325.46,0.00),v40,z0,tPen\WObj:=wPaper;
    MoveL Offs(pOrigin,265.51,324.41,0.00),v40,z0,tPen\WObj:=wPaper;
    MoveL Offs(pOrigin,268.70,324.41,0.00),v40,fine,tPen\WObj:=wPaper;
    MoveL Offs(pOrigin,268.70,324.41,6.00),v60,z5,tPen\WObj:=wPaper;
    MoveL Offs(pOrigin,267.85,323.35,6.00),vTravel,z5,tPen\WObj:=wPaper;
    MoveL Offs(pOrigin,267.85,323.35,0.00),v60,z0,tPen\WObj:=wPaper;
    MoveL Offs(pOrigin,264.66,323.35,0.00),v40,z0,tPen\WObj:=wPaper;
    MoveL Offs(pOrigin,265.51,323.11,0.00),v40,z0,tPen\WObj:=wPaper;
    MoveL Offs(pOrigin,266.36,323.96,0.00),v40,z0,tPen\WObj:=wPaper;
    MoveL Offs(pOrigin,265.51,323.11,0.00),v40,fine,tPen\WObj:=wPaper;
    MoveL Offs(pOrigin,265.51,323.11,6.00),v60,z5,tPen\WObj:=wPaper;
    MoveL Offs(pOrigin,266.79,322.30,6.00),vTravel,z5,tPen\WObj:=wPaper;
    MoveL Offs(pOrigin,266.79,322.30,0.00),v60,z0,tPen\WObj:=wPaper;
    MoveL Offs(pOrigin,260.84,322.30,0.00),v40,z0,tPen\WObj:=wPaper;
    MoveL Offs(pOrigin,260.41,322.69,0.00),v40,z0,tPen\WObj:=wPaper;
    MoveL Offs(pOrigin,260.84,323.11,0.00),v40,z0,tPen\WObj:=wPaper;
    MoveL Offs(pOrigin,260.41,322.69,0.00),v40,z0,tPen\WObj:=wPaper;
    MoveL Offs(pOrigin,260.85,321.62,0.00),v40,z0,tPen\WObj:=wPaper;
    MoveL Offs(pOrigin,260.85,320.56,0.00),v40,fine,tPen\WObj:=wPaper;
    MoveL Offs(pOrigin,260.85,320.56,6.00),v60,z5,tPen\WObj:=wPaper;
    MoveL Offs(pOrigin,261.48,321.62,6.00),vTravel,z5,tPen\WObj:=wPaper;
    MoveL Offs(pOrigin,261.48,321.62,0.00),v60,z0,tPen\WObj:=wPaper;
  ENDPROC

  PROC DrawPart238()
    MoveL Offs(pOrigin,262.33,322.48,0.00),v40,z0,tPen\WObj:=wPaper;
    MoveL Offs(pOrigin,261.48,321.62,0.00),v40,fine,tPen\WObj:=wPaper;
    MoveL Offs(pOrigin,261.48,321.62,6.00),v60,z5,tPen\WObj:=wPaper;
    MoveL Offs(pOrigin,263.10,324.63,6.00),vTravel,z5,tPen\WObj:=wPaper;
    MoveL Offs(pOrigin,263.10,324.63,0.00),v60,z0,tPen\WObj:=wPaper;
    MoveL Offs(pOrigin,251.23,312.76,0.00),v40,fine,tPen\WObj:=wPaper;
    MoveL Offs(pOrigin,251.23,312.76,6.00),v60,z5,tPen\WObj:=wPaper;
    MoveL Offs(pOrigin,252.19,311.07,6.00),vTravel,z5,tPen\WObj:=wPaper;
    MoveL Offs(pOrigin,252.19,311.07,0.00),v60,z0,tPen\WObj:=wPaper;
    MoveL Offs(pOrigin,236.26,327.00,0.00),v40,z0,tPen\WObj:=wPaper;
    MoveL Offs(pOrigin,236.75,326.64,0.00),v40,z0,tPen\WObj:=wPaper;
    MoveL Offs(pOrigin,237.95,327.85,0.00),v40,fine,tPen\WObj:=wPaper;
    MoveL Offs(pOrigin,237.95,327.85,6.00),v60,z5,tPen\WObj:=wPaper;
    MoveL Offs(pOrigin,236.56,328.20,6.00),vTravel,z5,tPen\WObj:=wPaper;
    MoveL Offs(pOrigin,236.56,328.20,0.00),v60,z0,tPen\WObj:=wPaper;
    MoveL Offs(pOrigin,253.69,311.07,0.00),v40,z0,tPen\WObj:=wPaper;
    MoveL Offs(pOrigin,254.44,311.82,0.00),v40,z0,tPen\WObj:=wPaper;
    MoveL Offs(pOrigin,236.25,330.00,0.00),v40,fine,tPen\WObj:=wPaper;
    MoveL Offs(pOrigin,236.25,330.00,6.00),v60,z5,tPen\WObj:=wPaper;
    MoveL Offs(pOrigin,237.46,330.76,6.00),vTravel,z5,tPen\WObj:=wPaper;
    MoveL Offs(pOrigin,237.46,330.76,0.00),v60,z0,tPen\WObj:=wPaper;
    MoveL Offs(pOrigin,237.25,331.19,0.00),v40,z0,tPen\WObj:=wPaper;
    MoveL Offs(pOrigin,237.46,330.76,0.00),v40,fine,tPen\WObj:=wPaper;
    MoveL Offs(pOrigin,237.46,330.76,6.00),v60,z5,tPen\WObj:=wPaper;
    MoveL Offs(pOrigin,238.11,332.49,6.00),vTravel,z5,tPen\WObj:=wPaper;
    MoveL Offs(pOrigin,238.11,332.49,0.00),v60,z0,tPen\WObj:=wPaper;
    MoveL Offs(pOrigin,239.16,333.54,0.00),v40,fine,tPen\WObj:=wPaper;
    MoveL Offs(pOrigin,239.16,333.54,6.00),v60,z5,tPen\WObj:=wPaper;
    MoveL Offs(pOrigin,239.08,336.13,6.00),vTravel,z5,tPen\WObj:=wPaper;
    MoveL Offs(pOrigin,239.08,336.13,0.00),v60,z0,tPen\WObj:=wPaper;
    MoveL Offs(pOrigin,234.72,340.49,0.00),v40,z0,tPen\WObj:=wPaper;
    MoveL Offs(pOrigin,235.29,340.12,0.00),v40,z0,tPen\WObj:=wPaper;
    MoveL Offs(pOrigin,233.94,338.77,0.00),v40,z0,tPen\WObj:=wPaper;
    MoveL Offs(pOrigin,234.43,337.79,0.00),v40,z0,tPen\WObj:=wPaper;
    MoveL Offs(pOrigin,231.73,340.50,0.00),v40,z0,tPen\WObj:=wPaper;
    MoveL Offs(pOrigin,232.44,340.26,0.00),v40,z0,tPen\WObj:=wPaper;
    MoveL Offs(pOrigin,230.64,338.46,0.00),v40,z0,tPen\WObj:=wPaper;
    MoveL Offs(pOrigin,231.44,337.80,0.00),v40,z0,tPen\WObj:=wPaper;
    MoveL Offs(pOrigin,229.18,340.05,0.00),v40,z0,tPen\WObj:=wPaper;
    MoveL Offs(pOrigin,229.30,340.10,0.00),v40,z0,tPen\WObj:=wPaper;
    MoveL Offs(pOrigin,222.24,333.04,0.00),v40,z0,tPen\WObj:=wPaper;
    MoveL Offs(pOrigin,222.16,333.52,0.00),v40,z0,tPen\WObj:=wPaper;
    MoveL Offs(pOrigin,222.80,332.75,0.00),v40,z0,tPen\WObj:=wPaper;
    MoveL Offs(pOrigin,224.93,332.46,0.00),v40,z0,tPen\WObj:=wPaper;
    MoveL Offs(pOrigin,225.35,331.83,0.00),v40,z0,tPen\WObj:=wPaper;
    MoveL Offs(pOrigin,225.23,331.55,0.00),v40,z0,tPen\WObj:=wPaper;
    MoveL Offs(pOrigin,227.63,333.96,0.00),v40,z0,tPen\WObj:=wPaper;
    MoveL Offs(pOrigin,227.05,333.10,0.00),v40,z0,tPen\WObj:=wPaper;
    MoveL Offs(pOrigin,227.05,331.40,0.00),v40,z0,tPen\WObj:=wPaper;
    MoveL Offs(pOrigin,226.62,331.19,0.00),v40,z0,tPen\WObj:=wPaper;
    MoveL Offs(pOrigin,228.32,331.61,0.00),v40,z0,tPen\WObj:=wPaper;
    MoveL Offs(pOrigin,229.81,330.98,0.00),v40,z0,tPen\WObj:=wPaper;
    MoveL Offs(pOrigin,229.87,330.22,0.00),v40,z0,tPen\WObj:=wPaper;
    MoveL Offs(pOrigin,229.11,329.47,0.00),v40,z0,tPen\WObj:=wPaper;
    MoveL Offs(pOrigin,228.22,330.06,0.00),v40,z0,tPen\WObj:=wPaper;
    MoveL Offs(pOrigin,230.32,332.17,0.00),v40,z0,tPen\WObj:=wPaper;
    MoveL Offs(pOrigin,230.85,332.41,0.00),v40,z0,tPen\WObj:=wPaper;
    MoveL Offs(pOrigin,233.56,329.71,0.00),v40,z0,tPen\WObj:=wPaper;
    MoveL Offs(pOrigin,233.21,329.91,0.00),v40,z0,tPen\WObj:=wPaper;
    MoveL Offs(pOrigin,232.79,330.55,0.00),v40,z0,tPen\WObj:=wPaper;
    MoveL Offs(pOrigin,233.21,329.91,0.00),v40,z0,tPen\WObj:=wPaper;
    MoveL Offs(pOrigin,233.64,329.06,0.00),v40,z0,tPen\WObj:=wPaper;
    MoveL Offs(pOrigin,233.43,329.49,0.00),v40,z0,tPen\WObj:=wPaper;
    MoveL Offs(pOrigin,233.64,329.06,0.00),v40,fine,tPen\WObj:=wPaper;
    MoveL Offs(pOrigin,233.64,329.06,6.00),v60,z5,tPen\WObj:=wPaper;
    MoveL Offs(pOrigin,232.36,329.27,6.00),vTravel,z5,tPen\WObj:=wPaper;
    MoveL Offs(pOrigin,232.36,329.27,0.00),v60,z0,tPen\WObj:=wPaper;
    MoveL Offs(pOrigin,232.15,329.70,0.00),v40,z0,tPen\WObj:=wPaper;
    MoveL Offs(pOrigin,232.36,329.27,0.00),v40,z0,tPen\WObj:=wPaper;
    MoveL Offs(pOrigin,231.31,328.96,0.00),v40,z0,tPen\WObj:=wPaper;
    MoveL Offs(pOrigin,222.15,338.13,0.00),v40,z0,tPen\WObj:=wPaper;
    MoveL Offs(pOrigin,222.16,337.08,0.00),v40,z0,tPen\WObj:=wPaper;
    MoveL Offs(pOrigin,225.14,337.08,0.00),v40,z0,tPen\WObj:=wPaper;
    MoveL Offs(pOrigin,225.99,336.92,0.00),v40,z0,tPen\WObj:=wPaper;
    MoveL Offs(pOrigin,222.80,336.71,0.00),v40,z0,tPen\WObj:=wPaper;
    MoveL Offs(pOrigin,222.02,336.29,0.00),v40,z0,tPen\WObj:=wPaper;
    MoveL Offs(pOrigin,221.95,335.86,0.00),v40,z0,tPen\WObj:=wPaper;
    MoveL Offs(pOrigin,221.95,335.86,0.00),v40,z0,tPen\WObj:=wPaper;
    MoveL Offs(pOrigin,217.91,335.23,0.00),v40,fine,tPen\WObj:=wPaper;
    MoveL Offs(pOrigin,217.91,335.23,6.00),v60,z5,tPen\WObj:=wPaper;
    MoveL Offs(pOrigin,219.40,336.02,6.00),vTravel,z5,tPen\WObj:=wPaper;
    MoveL Offs(pOrigin,219.40,336.02,0.00),v60,z0,tPen\WObj:=wPaper;
    MoveL Offs(pOrigin,221.31,336.02,0.00),v40,z0,tPen\WObj:=wPaper;
    MoveL Offs(pOrigin,221.77,335.01,0.00),v40,z0,tPen\WObj:=wPaper;
    MoveL Offs(pOrigin,221.77,333.95,0.00),v40,z0,tPen\WObj:=wPaper;
    MoveL Offs(pOrigin,222.83,333.74,0.00),v40,z0,tPen\WObj:=wPaper;
    MoveL Offs(pOrigin,222.83,334.80,0.00),v40,z0,tPen\WObj:=wPaper;
    MoveL Offs(pOrigin,222.59,335.65,0.00),v40,z0,tPen\WObj:=wPaper;
    MoveL Offs(pOrigin,224.71,335.86,0.00),v40,fine,tPen\WObj:=wPaper;
    MoveL Offs(pOrigin,224.71,335.86,6.00),v60,z5,tPen\WObj:=wPaper;
    MoveL Offs(pOrigin,225.99,336.92,6.00),vTravel,z5,tPen\WObj:=wPaper;
    MoveL Offs(pOrigin,225.99,336.92,0.00),v60,z0,tPen\WObj:=wPaper;
    MoveL Offs(pOrigin,226.84,337.35,0.00),v40,z0,tPen\WObj:=wPaper;
    MoveL Offs(pOrigin,226.62,338.14,0.00),v40,z0,tPen\WObj:=wPaper;
    MoveL Offs(pOrigin,224.50,338.14,0.00),v40,z0,tPen\WObj:=wPaper;
    MoveL Offs(pOrigin,224.39,338.87,0.00),v40,z0,tPen\WObj:=wPaper;
    MoveL Offs(pOrigin,229.20,334.06,0.00),v40,z0,tPen\WObj:=wPaper;
    MoveL Offs(pOrigin,228.53,334.86,0.00),v40,z0,tPen\WObj:=wPaper;
    MoveL Offs(pOrigin,230.49,336.81,0.00),v40,fine,tPen\WObj:=wPaper;
    MoveL Offs(pOrigin,230.49,336.81,6.00),v60,z5,tPen\WObj:=wPaper;
    MoveL Offs(pOrigin,231.83,336.67,6.00),vTravel,z5,tPen\WObj:=wPaper;
    MoveL Offs(pOrigin,231.83,336.67,0.00),v60,z0,tPen\WObj:=wPaper;
    MoveL Offs(pOrigin,230.03,334.86,0.00),v40,fine,tPen\WObj:=wPaper;
    MoveL Offs(pOrigin,230.03,334.86,6.00),v60,z5,tPen\WObj:=wPaper;
    MoveL Offs(pOrigin,229.42,332.76,6.00),vTravel,z5,tPen\WObj:=wPaper;
    MoveL Offs(pOrigin,229.42,332.76,0.00),v60,z0,tPen\WObj:=wPaper;
    MoveL Offs(pOrigin,227.32,330.66,0.00),v40,z0,tPen\WObj:=wPaper;
    MoveL Offs(pOrigin,227.69,330.74,0.00),v40,z0,tPen\WObj:=wPaper;
    MoveL Offs(pOrigin,228.75,330.74,0.00),v40,z0,tPen\WObj:=wPaper;
    MoveL Offs(pOrigin,228.11,331.61,0.00),v40,z0,tPen\WObj:=wPaper;
    MoveL Offs(pOrigin,228.11,332.68,0.00),v40,z0,tPen\WObj:=wPaper;
    MoveL Offs(pOrigin,228.54,332.86,0.00),v40,z0,tPen\WObj:=wPaper;
    MoveL Offs(pOrigin,224.08,332.86,0.00),v40,z0,tPen\WObj:=wPaper;
    MoveL Offs(pOrigin,223.43,332.74,0.00),v40,z0,tPen\WObj:=wPaper;
    MoveL Offs(pOrigin,227.79,337.10,0.00),v40,fine,tPen\WObj:=wPaper;
    MoveL Offs(pOrigin,227.79,337.10,6.00),v60,z5,tPen\WObj:=wPaper;
    MoveL Offs(pOrigin,228.99,336.81,6.00),vTravel,z5,tPen\WObj:=wPaper;
    MoveL Offs(pOrigin,228.99,336.81,0.00),v60,z0,tPen\WObj:=wPaper;
    MoveL Offs(pOrigin,224.33,332.15,0.00),v40,fine,tPen\WObj:=wPaper;
    MoveL Offs(pOrigin,224.33,332.15,6.00),v60,z5,tPen\WObj:=wPaper;
  ENDPROC

  PROC DrawPart239()
    MoveL Offs(pOrigin,225.78,331.80,6.00),vTravel,z5,tPen\WObj:=wPaper;
    MoveL Offs(pOrigin,225.78,331.80,0.00),v60,z0,tPen\WObj:=wPaper;
    MoveL Offs(pOrigin,229.39,331.80,0.00),v40,fine,tPen\WObj:=wPaper;
    MoveL Offs(pOrigin,229.39,331.80,6.00),v60,z5,tPen\WObj:=wPaper;
    MoveL Offs(pOrigin,230.66,331.19,6.00),vTravel,z5,tPen\WObj:=wPaper;
    MoveL Offs(pOrigin,230.66,331.19,0.00),v60,z0,tPen\WObj:=wPaper;
    MoveL Offs(pOrigin,229.81,330.55,0.00),v40,z0,tPen\WObj:=wPaper;
    MoveL Offs(pOrigin,230.73,329.06,0.00),v40,z0,tPen\WObj:=wPaper;
    MoveL Offs(pOrigin,231.30,327.15,0.00),v40,z0,tPen\WObj:=wPaper;
    MoveL Offs(pOrigin,231.09,323.75,0.00),v40,z0,tPen\WObj:=wPaper;
    MoveL Offs(pOrigin,231.51,323.47,0.00),v40,z0,tPen\WObj:=wPaper;
    MoveL Offs(pOrigin,232.86,325.45,0.00),v40,z0,tPen\WObj:=wPaper;
    MoveL Offs(pOrigin,233.21,327.15,0.00),v40,z0,tPen\WObj:=wPaper;
    MoveL Offs(pOrigin,232.93,328.42,0.00),v40,z0,tPen\WObj:=wPaper;
    MoveL Offs(pOrigin,231.44,330.34,0.00),v40,z0,tPen\WObj:=wPaper;
    MoveL Offs(pOrigin,231.30,331.19,0.00),v40,fine,tPen\WObj:=wPaper;
    MoveL Offs(pOrigin,231.30,331.19,6.00),v60,z5,tPen\WObj:=wPaper;
    MoveL Offs(pOrigin,230.45,329.27,6.00),vTravel,z5,tPen\WObj:=wPaper;
    MoveL Offs(pOrigin,230.45,329.27,0.00),v60,z0,tPen\WObj:=wPaper;
    MoveL Offs(pOrigin,230.02,329.70,0.00),v40,z0,tPen\WObj:=wPaper;
    MoveL Offs(pOrigin,230.45,329.27,0.00),v40,z0,tPen\WObj:=wPaper;
    MoveL Offs(pOrigin,230.76,328.12,0.00),v40,z0,tPen\WObj:=wPaper;
    MoveL Offs(pOrigin,230.01,327.37,0.00),v40,z0,tPen\WObj:=wPaper;
    MoveL Offs(pOrigin,231.05,326.93,0.00),v40,z0,tPen\WObj:=wPaper;
    MoveL Offs(pOrigin,230.15,326.02,0.00),v40,z0,tPen\WObj:=wPaper;
    MoveL Offs(pOrigin,231.05,325.43,0.00),v40,z0,tPen\WObj:=wPaper;
    MoveL Offs(pOrigin,229.55,323.93,0.00),v40,fine,tPen\WObj:=wPaper;
    MoveL Offs(pOrigin,229.55,323.93,6.00),v60,z5,tPen\WObj:=wPaper;
    MoveL Offs(pOrigin,228.92,328.37,6.00),vTravel,z5,tPen\WObj:=wPaper;
    MoveL Offs(pOrigin,228.92,328.37,0.00),v60,z0,tPen\WObj:=wPaper;
    MoveL Offs(pOrigin,245.60,311.69,0.00),v40,z0,tPen\WObj:=wPaper;
    MoveL Offs(pOrigin,245.11,311.64,0.00),v40,z0,tPen\WObj:=wPaper;
    MoveL Offs(pOrigin,244.33,312.06,0.00),v40,z0,tPen\WObj:=wPaper;
    MoveL Offs(pOrigin,243.84,313.55,0.00),v40,z0,tPen\WObj:=wPaper;
    MoveL Offs(pOrigin,243.84,315.25,0.00),v40,z0,tPen\WObj:=wPaper;
    MoveL Offs(pOrigin,244.26,316.74,0.00),v40,z0,tPen\WObj:=wPaper;
    MoveL Offs(pOrigin,243.77,318.23,0.00),v40,z0,tPen\WObj:=wPaper;
    MoveL Offs(pOrigin,244.05,318.44,0.00),v40,fine,tPen\WObj:=wPaper;
    MoveL Offs(pOrigin,244.05,318.44,6.00),v60,z5,tPen\WObj:=wPaper;
    MoveL Offs(pOrigin,246.06,317.80,6.00),vTravel,z5,tPen\WObj:=wPaper;
    MoveL Offs(pOrigin,246.06,317.80,0.00),v60,z0,tPen\WObj:=wPaper;
    MoveL Offs(pOrigin,246.06,320.35,0.00),v40,z0,tPen\WObj:=wPaper;
    MoveL Offs(pOrigin,246.60,321.20,0.00),v40,z0,tPen\WObj:=wPaper;
    MoveL Offs(pOrigin,247.02,321.41,0.00),v40,z0,tPen\WObj:=wPaper;
    MoveL Offs(pOrigin,246.60,321.20,0.00),v40,z0,tPen\WObj:=wPaper;
    MoveL Offs(pOrigin,247.12,320.77,0.00),v40,z0,tPen\WObj:=wPaper;
    MoveL Offs(pOrigin,247.12,318.86,0.00),v40,z0,tPen\WObj:=wPaper;
    MoveL Offs(pOrigin,247.45,318.86,0.00),v40,z0,tPen\WObj:=wPaper;
    MoveL Offs(pOrigin,248.94,319.08,0.00),v40,z0,tPen\WObj:=wPaper;
    MoveL Offs(pOrigin,249.79,318.65,0.00),v40,z0,tPen\WObj:=wPaper;
    MoveL Offs(pOrigin,252.12,319.08,0.00),v40,fine,tPen\WObj:=wPaper;
    MoveL Offs(pOrigin,252.12,319.08,6.00),v60,z5,tPen\WObj:=wPaper;
    MoveL Offs(pOrigin,250.29,318.65,6.00),vTravel,z5,tPen\WObj:=wPaper;
    MoveL Offs(pOrigin,250.29,318.65,0.00),v60,z0,tPen\WObj:=wPaper;
    MoveL Offs(pOrigin,250.29,320.35,0.00),v40,fine,tPen\WObj:=wPaper;
    MoveL Offs(pOrigin,250.29,320.35,6.00),v60,z5,tPen\WObj:=wPaper;
    MoveL Offs(pOrigin,251.49,315.96,6.00),vTravel,z5,tPen\WObj:=wPaper;
    MoveL Offs(pOrigin,251.49,315.96,0.00),v60,z0,tPen\WObj:=wPaper;
    MoveL Offs(pOrigin,272.31,315.96,0.00),v40,fine,tPen\WObj:=wPaper;
    MoveL Offs(pOrigin,272.31,315.96,6.00),v60,z5,tPen\WObj:=wPaper;
    MoveL Offs(pOrigin,274.01,315.25,6.00),vTravel,z5,tPen\WObj:=wPaper;
    MoveL Offs(pOrigin,274.01,315.25,0.00),v60,z0,tPen\WObj:=wPaper;
    MoveL Offs(pOrigin,274.23,315.67,0.00),v40,z0,tPen\WObj:=wPaper;
    MoveL Offs(pOrigin,274.01,315.25,0.00),v40,fine,tPen\WObj:=wPaper;
    MoveL Offs(pOrigin,274.01,315.25,6.00),v60,z5,tPen\WObj:=wPaper;
    MoveL Offs(pOrigin,274.86,311.74,6.00),vTravel,z5,tPen\WObj:=wPaper;
    MoveL Offs(pOrigin,274.86,311.74,0.00),v60,z0,tPen\WObj:=wPaper;
    MoveL Offs(pOrigin,264.24,311.74,0.00),v40,fine,tPen\WObj:=wPaper;
    MoveL Offs(pOrigin,264.24,311.74,6.00),v60,z5,tPen\WObj:=wPaper;
    MoveL Offs(pOrigin,263.18,310.68,6.00),vTravel,z5,tPen\WObj:=wPaper;
    MoveL Offs(pOrigin,263.18,310.68,0.00),v60,z0,tPen\WObj:=wPaper;
    MoveL Offs(pOrigin,278.05,310.68,0.00),v40,fine,tPen\WObj:=wPaper;
    MoveL Offs(pOrigin,278.05,310.68,6.00),v60,z5,tPen\WObj:=wPaper;
    MoveL Offs(pOrigin,277.62,309.30,6.00),vTravel,z5,tPen\WObj:=wPaper;
    MoveL Offs(pOrigin,277.62,309.30,0.00),v60,z0,tPen\WObj:=wPaper;
    MoveL Offs(pOrigin,276.56,309.30,0.00),v40,z0,tPen\WObj:=wPaper;
    MoveL Offs(pOrigin,276.35,309.73,0.00),v40,z0,tPen\WObj:=wPaper;
    MoveL Offs(pOrigin,276.69,308.66,0.00),v40,z0,tPen\WObj:=wPaper;
    MoveL Offs(pOrigin,276.69,301.86,0.00),v40,z0,tPen\WObj:=wPaper;
    MoveL Offs(pOrigin,276.56,301.18,0.00),v40,z0,tPen\WObj:=wPaper;
    MoveL Offs(pOrigin,281.45,301.18,0.00),v40,z0,tPen\WObj:=wPaper;
    MoveL Offs(pOrigin,281.24,300.12,0.00),v40,z0,tPen\WObj:=wPaper;
    MoveL Offs(pOrigin,277.20,300.12,0.00),v40,z0,tPen\WObj:=wPaper;
    MoveL Offs(pOrigin,276.81,299.50,0.00),v40,z0,tPen\WObj:=wPaper;
    MoveL Offs(pOrigin,282.22,304.91,0.00),v40,z0,tPen\WObj:=wPaper;
    MoveL Offs(pOrigin,282.96,304.17,0.00),v40,z0,tPen\WObj:=wPaper;
    MoveL Offs(pOrigin,277.26,298.46,0.00),v40,z0,tPen\WObj:=wPaper;
    MoveL Offs(pOrigin,277.62,298.89,0.00),v40,z0,tPen\WObj:=wPaper;
    MoveL Offs(pOrigin,276.56,299.52,0.00),v40,z0,tPen\WObj:=wPaper;
    MoveL Offs(pOrigin,275.43,301.86,0.00),v40,z0,tPen\WObj:=wPaper;
    MoveL Offs(pOrigin,275.92,302.64,0.00),v40,z0,tPen\WObj:=wPaper;
    MoveL Offs(pOrigin,276.77,302.71,0.00),v40,z0,tPen\WObj:=wPaper;
    MoveL Offs(pOrigin,276.77,302.71,0.00),v40,z0,tPen\WObj:=wPaper;
    MoveL Offs(pOrigin,278.69,301.37,0.00),v40,z0,tPen\WObj:=wPaper;
    MoveL Offs(pOrigin,279.96,300.94,0.00),v40,z0,tPen\WObj:=wPaper;
    MoveL Offs(pOrigin,280.60,300.16,0.00),v40,fine,tPen\WObj:=wPaper;
    MoveL Offs(pOrigin,280.60,300.16,6.00),v60,z5,tPen\WObj:=wPaper;
    MoveL Offs(pOrigin,281.45,299.06,6.00),vTravel,z5,tPen\WObj:=wPaper;
    MoveL Offs(pOrigin,281.45,299.06,0.00),v60,z0,tPen\WObj:=wPaper;
    MoveL Offs(pOrigin,277.84,299.06,0.00),v40,fine,tPen\WObj:=wPaper;
    MoveL Offs(pOrigin,277.84,299.06,6.00),v60,z5,tPen\WObj:=wPaper;
    MoveL Offs(pOrigin,278.48,298.01,6.00),vTravel,z5,tPen\WObj:=wPaper;
    MoveL Offs(pOrigin,278.48,298.01,0.00),v60,z0,tPen\WObj:=wPaper;
    MoveL Offs(pOrigin,282.09,298.01,0.00),v40,z0,tPen\WObj:=wPaper;
    MoveL Offs(pOrigin,281.88,296.95,0.00),v40,z0,tPen\WObj:=wPaper;
    MoveL Offs(pOrigin,278.69,296.95,0.00),v40,z0,tPen\WObj:=wPaper;
    MoveL Offs(pOrigin,278.15,296.36,0.00),v40,z0,tPen\WObj:=wPaper;
    MoveL Offs(pOrigin,283.56,301.77,0.00),v40,z0,tPen\WObj:=wPaper;
    MoveL Offs(pOrigin,282.81,302.52,0.00),v40,z0,tPen\WObj:=wPaper;
    MoveL Offs(pOrigin,277.70,297.41,0.00),v40,z0,tPen\WObj:=wPaper;
    MoveL Offs(pOrigin,277.10,296.62,0.00),v40,z0,tPen\WObj:=wPaper;
    MoveL Offs(pOrigin,302.05,271.67,0.00),v40,z0,tPen\WObj:=wPaper;
    MoveL Offs(pOrigin,301.42,271.48,0.00),v40,z0,tPen\WObj:=wPaper;
    MoveL Offs(pOrigin,301.00,272.11,0.00),v40,z0,tPen\WObj:=wPaper;
    MoveL Offs(pOrigin,301.42,271.48,0.00),v40,z0,tPen\WObj:=wPaper;
    MoveL Offs(pOrigin,301.29,271.72,0.00),v40,z0,tPen\WObj:=wPaper;
    MoveL Offs(pOrigin,300.24,270.66,0.00),v40,z0,tPen\WObj:=wPaper;
    MoveL Offs(pOrigin,299.64,271.56,0.00),v40,z0,tPen\WObj:=wPaper;
    MoveL Offs(pOrigin,300.69,272.61,0.00),v40,z0,tPen\WObj:=wPaper;
    MoveL Offs(pOrigin,300.79,272.54,0.00),v40,z0,tPen\WObj:=wPaper;
  ENDPROC

  PROC DrawPart240()
    MoveL Offs(pOrigin,300.36,273.17,0.00),v40,z0,tPen\WObj:=wPaper;
    MoveL Offs(pOrigin,300.79,272.54,0.00),v40,fine,tPen\WObj:=wPaper;
    MoveL Offs(pOrigin,300.79,272.54,6.00),v60,z5,tPen\WObj:=wPaper;
    MoveL Offs(pOrigin,299.73,271.69,6.00),vTravel,z5,tPen\WObj:=wPaper;
    MoveL Offs(pOrigin,299.73,271.69,0.00),v60,z0,tPen\WObj:=wPaper;
    MoveL Offs(pOrigin,299.30,272.33,0.00),v40,z0,tPen\WObj:=wPaper;
    MoveL Offs(pOrigin,299.73,271.69,0.00),v40,fine,tPen\WObj:=wPaper;
    MoveL Offs(pOrigin,299.73,271.69,6.00),v60,z5,tPen\WObj:=wPaper;
    MoveL Offs(pOrigin,300.69,269.62,6.00),vTravel,z5,tPen\WObj:=wPaper;
    MoveL Offs(pOrigin,300.69,269.62,0.00),v60,z0,tPen\WObj:=wPaper;
    MoveL Offs(pOrigin,301.89,270.82,0.00),v40,z0,tPen\WObj:=wPaper;
    MoveL Offs(pOrigin,301.85,270.62,0.00),v40,z0,tPen\WObj:=wPaper;
    MoveL Offs(pOrigin,301.64,271.05,0.00),v40,z0,tPen\WObj:=wPaper;
    MoveL Offs(pOrigin,301.85,270.62,0.00),v40,z0,tPen\WObj:=wPaper;
    MoveL Offs(pOrigin,302.48,269.92,0.00),v40,z0,tPen\WObj:=wPaper;
    MoveL Offs(pOrigin,301.13,268.57,0.00),v40,fine,tPen\WObj:=wPaper;
    MoveL Offs(pOrigin,301.13,268.57,6.00),v60,z5,tPen\WObj:=wPaper;
    MoveL Offs(pOrigin,301.28,267.22,6.00),vTravel,z5,tPen\WObj:=wPaper;
    MoveL Offs(pOrigin,301.28,267.22,0.00),v60,z0,tPen\WObj:=wPaper;
    MoveL Offs(pOrigin,302.63,268.57,0.00),v40,z0,tPen\WObj:=wPaper;
    MoveL Offs(pOrigin,303.10,269.12,0.00),v40,z0,tPen\WObj:=wPaper;
    MoveL Offs(pOrigin,277.86,294.37,0.00),v40,fine,tPen\WObj:=wPaper;
    MoveL Offs(pOrigin,277.86,294.37,6.00),v60,z5,tPen\WObj:=wPaper;
    MoveL Offs(pOrigin,279.75,293.78,6.00),vTravel,z5,tPen\WObj:=wPaper;
    MoveL Offs(pOrigin,279.75,293.78,0.00),v60,z0,tPen\WObj:=wPaper;
    MoveL Offs(pOrigin,283.79,293.78,0.00),v40,fine,tPen\WObj:=wPaper;
    MoveL Offs(pOrigin,283.79,293.78,6.00),v60,z5,tPen\WObj:=wPaper;
    MoveL Offs(pOrigin,284.85,292.73,6.00),vTravel,z5,tPen\WObj:=wPaper;
    MoveL Offs(pOrigin,284.85,292.73,0.00),v60,z0,tPen\WObj:=wPaper;
    MoveL Offs(pOrigin,280.18,292.73,0.00),v40,z0,tPen\WObj:=wPaper;
    MoveL Offs(pOrigin,280.91,293.15,0.00),v40,z0,tPen\WObj:=wPaper;
    MoveL Offs(pOrigin,280.91,296.76,0.00),v40,fine,tPen\WObj:=wPaper;
    MoveL Offs(pOrigin,280.91,296.76,6.00),v60,z5,tPen\WObj:=wPaper;
    MoveL Offs(pOrigin,280.39,295.27,6.00),vTravel,z5,tPen\WObj:=wPaper;
    MoveL Offs(pOrigin,280.39,295.27,0.00),v60,z0,tPen\WObj:=wPaper;
    MoveL Offs(pOrigin,280.60,294.42,0.00),v40,z0,tPen\WObj:=wPaper;
    MoveL Offs(pOrigin,281.66,293.79,0.00),v40,fine,tPen\WObj:=wPaper;
    MoveL Offs(pOrigin,281.66,293.79,6.00),v60,z5,tPen\WObj:=wPaper;
    MoveL Offs(pOrigin,281.97,290.81,6.00),vTravel,z5,tPen\WObj:=wPaper;
    MoveL Offs(pOrigin,281.97,290.81,0.00),v60,z0,tPen\WObj:=wPaper;
    MoveL Offs(pOrigin,281.97,284.22,0.00),v40,fine,tPen\WObj:=wPaper;
    MoveL Offs(pOrigin,281.97,284.22,6.00),v60,z5,tPen\WObj:=wPaper;
    MoveL Offs(pOrigin,283.02,282.95,6.00),vTravel,z5,tPen\WObj:=wPaper;
    MoveL Offs(pOrigin,283.02,282.95,0.00),v60,z0,tPen\WObj:=wPaper;
    MoveL Offs(pOrigin,283.02,286.14,0.00),v40,fine,tPen\WObj:=wPaper;
    MoveL Offs(pOrigin,283.02,286.14,6.00),v60,z5,tPen\WObj:=wPaper;
    MoveL Offs(pOrigin,284.08,283.16,6.00),vTravel,z5,tPen\WObj:=wPaper;
    MoveL Offs(pOrigin,284.08,283.16,0.00),v60,z0,tPen\WObj:=wPaper;
    MoveL Offs(pOrigin,284.08,281.68,0.00),v40,fine,tPen\WObj:=wPaper;
    MoveL Offs(pOrigin,284.08,281.68,6.00),v60,z5,tPen\WObj:=wPaper;
    MoveL Offs(pOrigin,282.73,282.10,6.00),vTravel,z5,tPen\WObj:=wPaper;
    MoveL Offs(pOrigin,282.73,282.10,0.00),v60,z0,tPen\WObj:=wPaper;
    MoveL Offs(pOrigin,282.51,282.52,0.00),v40,z0,tPen\WObj:=wPaper;
    MoveL Offs(pOrigin,282.73,282.10,0.00),v40,fine,tPen\WObj:=wPaper;
    MoveL Offs(pOrigin,282.73,282.10,6.00),v60,z5,tPen\WObj:=wPaper;
    MoveL Offs(pOrigin,286.19,281.46,6.00),vTravel,z5,tPen\WObj:=wPaper;
    MoveL Offs(pOrigin,286.19,281.46,0.00),v60,z0,tPen\WObj:=wPaper;
    MoveL Offs(pOrigin,286.19,279.97,0.00),v40,fine,tPen\WObj:=wPaper;
    MoveL Offs(pOrigin,286.19,279.97,6.00),v60,z5,tPen\WObj:=wPaper;
    MoveL Offs(pOrigin,288.67,286.14,6.00),vTravel,z5,tPen\WObj:=wPaper;
    MoveL Offs(pOrigin,288.67,286.14,0.00),v60,z0,tPen\WObj:=wPaper;
    MoveL Offs(pOrigin,289.10,285.50,0.00),v40,z0,tPen\WObj:=wPaper;
    MoveL Offs(pOrigin,290.16,285.71,0.00),v40,z0,tPen\WObj:=wPaper;
    MoveL Offs(pOrigin,290.16,285.50,0.00),v40,z0,tPen\WObj:=wPaper;
    MoveL Offs(pOrigin,290.16,285.50,0.00),v40,z0,tPen\WObj:=wPaper;
    MoveL Offs(pOrigin,293.35,286.14,0.00),v40,z0,tPen\WObj:=wPaper;
    MoveL Offs(pOrigin,293.14,285.71,0.00),v40,z0,tPen\WObj:=wPaper;
    MoveL Offs(pOrigin,293.35,286.14,0.00),v40,z0,tPen\WObj:=wPaper;
    MoveL Offs(pOrigin,293.14,285.71,0.00),v40,fine,tPen\WObj:=wPaper;
    MoveL Offs(pOrigin,293.14,285.71,6.00),v60,z5,tPen\WObj:=wPaper;
    MoveL Offs(pOrigin,293.58,286.99,6.00),vTravel,z5,tPen\WObj:=wPaper;
    MoveL Offs(pOrigin,293.58,286.99,0.00),v60,z0,tPen\WObj:=wPaper;
    MoveL Offs(pOrigin,293.58,288.69,0.00),v40,fine,tPen\WObj:=wPaper;
    MoveL Offs(pOrigin,293.58,288.69,6.00),v60,z5,tPen\WObj:=wPaper;
    MoveL Offs(pOrigin,292.53,288.05,6.00),vTravel,z5,tPen\WObj:=wPaper;
    MoveL Offs(pOrigin,292.53,288.05,0.00),v60,z0,tPen\WObj:=wPaper;
    MoveL Offs(pOrigin,292.53,286.99,0.00),v40,fine,tPen\WObj:=wPaper;
    MoveL Offs(pOrigin,292.53,286.99,6.00),v60,z5,tPen\WObj:=wPaper;
    MoveL Offs(pOrigin,294.64,287.41,6.00),vTravel,z5,tPen\WObj:=wPaper;
    MoveL Offs(pOrigin,294.64,287.41,0.00),v60,z0,tPen\WObj:=wPaper;
    MoveL Offs(pOrigin,294.64,289.54,0.00),v40,fine,tPen\WObj:=wPaper;
    MoveL Offs(pOrigin,294.64,289.54,6.00),v60,z5,tPen\WObj:=wPaper;
    MoveL Offs(pOrigin,296.75,294.64,6.00),vTravel,z5,tPen\WObj:=wPaper;
    MoveL Offs(pOrigin,296.75,294.64,0.00),v60,z0,tPen\WObj:=wPaper;
    MoveL Offs(pOrigin,296.75,281.46,0.00),v40,z0,tPen\WObj:=wPaper;
    MoveL Offs(pOrigin,297.81,281.68,0.00),v40,z0,tPen\WObj:=wPaper;
    MoveL Offs(pOrigin,297.81,283.38,0.00),v40,fine,tPen\WObj:=wPaper;
    MoveL Offs(pOrigin,297.81,283.38,6.00),v60,z5,tPen\WObj:=wPaper;
    MoveL Offs(pOrigin,293.35,283.38,6.00),vTravel,z5,tPen\WObj:=wPaper;
    MoveL Offs(pOrigin,293.35,283.38,0.00),v60,z0,tPen\WObj:=wPaper;
    MoveL Offs(pOrigin,293.56,283.80,0.00),v40,z0,tPen\WObj:=wPaper;
    MoveL Offs(pOrigin,293.35,283.38,0.00),v40,fine,tPen\WObj:=wPaper;
    MoveL Offs(pOrigin,293.35,283.38,6.00),v60,z5,tPen\WObj:=wPaper;
    MoveL Offs(pOrigin,288.89,286.56,6.00),vTravel,z5,tPen\WObj:=wPaper;
    MoveL Offs(pOrigin,288.89,286.56,0.00),v60,z0,tPen\WObj:=wPaper;
    MoveL Offs(pOrigin,288.46,286.21,0.00),v40,z0,tPen\WObj:=wPaper;
    MoveL Offs(pOrigin,287.61,286.35,0.00),v40,z0,tPen\WObj:=wPaper;
    MoveL Offs(pOrigin,285.91,287.27,0.00),v40,z0,tPen\WObj:=wPaper;
    MoveL Offs(pOrigin,284.42,288.90,0.00),v40,z0,tPen\WObj:=wPaper;
    MoveL Offs(pOrigin,284.00,289.96,0.00),v40,fine,tPen\WObj:=wPaper;
    MoveL Offs(pOrigin,284.00,289.96,6.00),v60,z5,tPen\WObj:=wPaper;
    MoveL Offs(pOrigin,288.67,296.76,6.00),vTravel,z5,tPen\WObj:=wPaper;
    MoveL Offs(pOrigin,288.67,296.76,0.00),v60,z0,tPen\WObj:=wPaper;
    MoveL Offs(pOrigin,288.04,297.40,0.00),v40,z0,tPen\WObj:=wPaper;
    MoveL Offs(pOrigin,288.67,296.76,0.00),v40,fine,tPen\WObj:=wPaper;
    MoveL Offs(pOrigin,288.67,296.76,6.00),v60,z5,tPen\WObj:=wPaper;
    MoveL Offs(pOrigin,289.10,299.10,6.00),vTravel,z5,tPen\WObj:=wPaper;
    MoveL Offs(pOrigin,289.10,299.10,0.00),v60,z0,tPen\WObj:=wPaper;
    MoveL Offs(pOrigin,286.98,299.95,0.00),v40,z0,tPen\WObj:=wPaper;
    MoveL Offs(pOrigin,286.55,299.52,0.00),v40,z0,tPen\WObj:=wPaper;
    MoveL Offs(pOrigin,286.55,298.46,0.00),v40,z0,tPen\WObj:=wPaper;
    MoveL Offs(pOrigin,290.38,295.77,0.00),v40,z0,tPen\WObj:=wPaper;
    MoveL Offs(pOrigin,291.23,295.70,0.00),v40,fine,tPen\WObj:=wPaper;
    MoveL Offs(pOrigin,291.23,295.70,6.00),v60,z5,tPen\WObj:=wPaper;
    MoveL Offs(pOrigin,286.54,298.78,6.00),vTravel,z5,tPen\WObj:=wPaper;
    MoveL Offs(pOrigin,286.54,298.78,0.00),v60,z0,tPen\WObj:=wPaper;
    MoveL Offs(pOrigin,294.51,306.75,0.00),v40,z0,tPen\WObj:=wPaper;
    MoveL Offs(pOrigin,295.50,306.60,0.00),v40,z0,tPen\WObj:=wPaper;
    MoveL Offs(pOrigin,284.53,317.57,0.00),v40,fine,tPen\WObj:=wPaper;
    MoveL Offs(pOrigin,284.53,317.57,6.00),v60,z5,tPen\WObj:=wPaper;
  ENDPROC

  PROC DrawPart241()
    MoveL Offs(pOrigin,283.61,319.75,6.00),vTravel,z5,tPen\WObj:=wPaper;
    MoveL Offs(pOrigin,283.61,319.75,0.00),v60,z0,tPen\WObj:=wPaper;
    MoveL Offs(pOrigin,286.77,322.90,0.00),v40,z0,tPen\WObj:=wPaper;
    MoveL Offs(pOrigin,286.98,322.90,0.00),v40,z0,tPen\WObj:=wPaper;
    MoveL Offs(pOrigin,286.34,323.54,0.00),v40,z0,tPen\WObj:=wPaper;
    MoveL Offs(pOrigin,286.98,322.90,0.00),v40,fine,tPen\WObj:=wPaper;
    MoveL Offs(pOrigin,286.98,322.90,6.00),v60,z5,tPen\WObj:=wPaper;
    MoveL Offs(pOrigin,287.19,320.35,6.00),vTravel,z5,tPen\WObj:=wPaper;
    MoveL Offs(pOrigin,287.19,320.35,0.00),v60,z0,tPen\WObj:=wPaper;
    MoveL Offs(pOrigin,286.98,320.77,0.00),v40,z0,tPen\WObj:=wPaper;
    MoveL Offs(pOrigin,287.19,320.35,0.00),v40,z0,tPen\WObj:=wPaper;
    MoveL Offs(pOrigin,287.40,320.18,0.00),v40,z0,tPen\WObj:=wPaper;
    MoveL Offs(pOrigin,284.64,320.18,0.00),v40,fine,tPen\WObj:=wPaper;
    MoveL Offs(pOrigin,284.64,320.18,6.00),v60,z5,tPen\WObj:=wPaper;
    MoveL Offs(pOrigin,281.37,321.99,6.00),vTravel,z5,tPen\WObj:=wPaper;
    MoveL Offs(pOrigin,281.37,321.99,0.00),v60,z0,tPen\WObj:=wPaper;
    MoveL Offs(pOrigin,284.38,324.99,0.00),v40,fine,tPen\WObj:=wPaper;
    MoveL Offs(pOrigin,284.38,324.99,6.00),v60,z5,tPen\WObj:=wPaper;
    MoveL Offs(pOrigin,289.00,319.16,6.00),vTravel,z5,tPen\WObj:=wPaper;
    MoveL Offs(pOrigin,289.00,319.16,0.00),v60,z0,tPen\WObj:=wPaper;
    MoveL Offs(pOrigin,287.20,317.36,0.00),v40,z0,tPen\WObj:=wPaper;
    MoveL Offs(pOrigin,288.04,317.02,0.00),v40,z0,tPen\WObj:=wPaper;
    MoveL Offs(pOrigin,289.74,317.02,0.00),v40,z0,tPen\WObj:=wPaper;
    MoveL Offs(pOrigin,290.49,316.17,0.00),v40,z0,tPen\WObj:=wPaper;
    MoveL Offs(pOrigin,288.39,314.07,0.00),v40,z0,tPen\WObj:=wPaper;
    MoveL Offs(pOrigin,289.10,313.85,0.00),v40,z0,tPen\WObj:=wPaper;
    MoveL Offs(pOrigin,291.44,313.85,0.00),v40,z0,tPen\WObj:=wPaper;
    MoveL Offs(pOrigin,290.80,314.19,0.00),v40,z0,tPen\WObj:=wPaper;
    MoveL Offs(pOrigin,291.65,311.85,0.00),v40,z0,tPen\WObj:=wPaper;
    MoveL Offs(pOrigin,291.65,311.85,0.00),v40,z0,tPen\WObj:=wPaper;
    MoveL Offs(pOrigin,292.71,311.64,0.00),v40,z0,tPen\WObj:=wPaper;
    MoveL Offs(pOrigin,293.02,311.24,0.00),v40,z0,tPen\WObj:=wPaper;
    MoveL Offs(pOrigin,287.16,305.38,0.00),v40,fine,tPen\WObj:=wPaper;
    MoveL Offs(pOrigin,287.16,305.38,6.00),v60,z5,tPen\WObj:=wPaper;
    MoveL Offs(pOrigin,288.67,305.69,6.00),vTravel,z5,tPen\WObj:=wPaper;
    MoveL Offs(pOrigin,288.67,305.69,0.00),v60,z0,tPen\WObj:=wPaper;
    MoveL Offs(pOrigin,288.46,306.11,0.00),v40,z0,tPen\WObj:=wPaper;
    MoveL Offs(pOrigin,288.67,305.69,0.00),v40,z0,tPen\WObj:=wPaper;
    MoveL Offs(pOrigin,289.10,304.84,0.00),v40,z0,tPen\WObj:=wPaper;
    MoveL Offs(pOrigin,288.89,305.26,0.00),v40,z0,tPen\WObj:=wPaper;
    MoveL Offs(pOrigin,289.10,304.84,0.00),v40,fine,tPen\WObj:=wPaper;
    MoveL Offs(pOrigin,289.10,304.84,6.00),v60,z5,tPen\WObj:=wPaper;
    MoveL Offs(pOrigin,292.29,306.54,6.00),vTravel,z5,tPen\WObj:=wPaper;
    MoveL Offs(pOrigin,292.29,306.54,0.00),v60,z0,tPen\WObj:=wPaper;
    MoveL Offs(pOrigin,292.08,307.81,0.00),v40,fine,tPen\WObj:=wPaper;
    MoveL Offs(pOrigin,292.08,307.81,6.00),v60,z5,tPen\WObj:=wPaper;
    MoveL Offs(pOrigin,293.35,308.57,6.00),vTravel,z5,tPen\WObj:=wPaper;
    MoveL Offs(pOrigin,293.35,308.57,0.00),v60,z0,tPen\WObj:=wPaper;
    MoveL Offs(pOrigin,288.89,308.57,0.00),v40,fine,tPen\WObj:=wPaper;
    MoveL Offs(pOrigin,288.89,308.57,6.00),v60,z5,tPen\WObj:=wPaper;
    MoveL Offs(pOrigin,288.68,310.68,6.00),vTravel,z5,tPen\WObj:=wPaper;
    MoveL Offs(pOrigin,288.68,310.68,0.00),v60,z0,tPen\WObj:=wPaper;
    MoveL Offs(pOrigin,287.61,310.68,0.00),v40,z0,tPen\WObj:=wPaper;
    MoveL Offs(pOrigin,286.58,310.77,0.00),v40,z0,tPen\WObj:=wPaper;
    MoveL Offs(pOrigin,291.24,315.43,0.00),v40,z0,tPen\WObj:=wPaper;
    MoveL Offs(pOrigin,290.80,316.10,0.00),v40,z0,tPen\WObj:=wPaper;
    MoveL Offs(pOrigin,290.38,316.52,0.00),v40,z0,tPen\WObj:=wPaper;
    MoveL Offs(pOrigin,290.80,316.10,0.00),v40,z0,tPen\WObj:=wPaper;
    MoveL Offs(pOrigin,290.38,315.96,0.00),v40,z0,tPen\WObj:=wPaper;
    MoveL Offs(pOrigin,288.68,315.96,0.00),v40,z0,tPen\WObj:=wPaper;
    MoveL Offs(pOrigin,288.04,316.74,0.00),v40,z0,tPen\WObj:=wPaper;
    MoveL Offs(pOrigin,287.83,317.16,0.00),v40,z0,tPen\WObj:=wPaper;
    MoveL Offs(pOrigin,288.04,316.74,0.00),v40,fine,tPen\WObj:=wPaper;
    MoveL Offs(pOrigin,288.04,316.74,6.00),v60,z5,tPen\WObj:=wPaper;
    MoveL Offs(pOrigin,286.19,314.41,6.00),vTravel,z5,tPen\WObj:=wPaper;
    MoveL Offs(pOrigin,286.19,314.41,0.00),v60,z0,tPen\WObj:=wPaper;
    MoveL Offs(pOrigin,297.15,303.45,0.00),v40,fine,tPen\WObj:=wPaper;
    MoveL Offs(pOrigin,297.15,303.45,6.00),v60,z5,tPen\WObj:=wPaper;
    MoveL Offs(pOrigin,298.07,296.55,6.00),vTravel,z5,tPen\WObj:=wPaper;
    MoveL Offs(pOrigin,298.07,296.55,0.00),v60,z0,tPen\WObj:=wPaper;
    MoveL Offs(pOrigin,286.05,308.57,0.00),v40,fine,tPen\WObj:=wPaper;
    MoveL Offs(pOrigin,286.05,308.57,6.00),v60,z5,tPen\WObj:=wPaper;
    MoveL Offs(pOrigin,286.06,307.07,6.00),vTravel,z5,tPen\WObj:=wPaper;
    MoveL Offs(pOrigin,286.06,307.07,0.00),v60,z0,tPen\WObj:=wPaper;
    MoveL Offs(pOrigin,298.23,294.90,0.00),v40,fine,tPen\WObj:=wPaper;
    MoveL Offs(pOrigin,298.23,294.90,6.00),v60,z5,tPen\WObj:=wPaper;
    MoveL Offs(pOrigin,287.15,300.88,6.00),vTravel,z5,tPen\WObj:=wPaper;
    MoveL Offs(pOrigin,287.15,300.88,0.00),v60,z0,tPen\WObj:=wPaper;
    MoveL Offs(pOrigin,286.10,299.83,0.00),v40,z0,tPen\WObj:=wPaper;
    MoveL Offs(pOrigin,286.55,299.95,0.00),v40,z0,tPen\WObj:=wPaper;
    MoveL Offs(pOrigin,286.55,300.38,0.00),v40,z0,tPen\WObj:=wPaper;
    MoveL Offs(pOrigin,285.91,301.01,0.00),v40,z0,tPen\WObj:=wPaper;
    MoveL Offs(pOrigin,285.49,301.01,0.00),v40,z0,tPen\WObj:=wPaper;
    MoveL Offs(pOrigin,285.65,300.88,0.00),v40,z0,tPen\WObj:=wPaper;
    MoveL Offs(pOrigin,286.40,301.63,0.00),v40,fine,tPen\WObj:=wPaper;
    MoveL Offs(pOrigin,286.40,301.63,6.00),v60,z5,tPen\WObj:=wPaper;
    MoveL Offs(pOrigin,281.47,305.66,6.00),vTravel,z5,tPen\WObj:=wPaper;
    MoveL Offs(pOrigin,281.47,305.66,0.00),v60,z0,tPen\WObj:=wPaper;
    MoveL Offs(pOrigin,276.21,300.40,0.00),v40,z0,tPen\WObj:=wPaper;
    MoveL Offs(pOrigin,275.60,299.62,0.00),v40,z0,tPen\WObj:=wPaper;
    MoveL Offs(pOrigin,300.69,274.52,0.00),v40,fine,tPen\WObj:=wPaper;
    MoveL Offs(pOrigin,300.69,274.52,6.00),v60,z5,tPen\WObj:=wPaper;
    MoveL Offs(pOrigin,300.53,276.17,6.00),vTravel,z5,tPen\WObj:=wPaper;
    MoveL Offs(pOrigin,300.53,276.17,0.00),v60,z0,tPen\WObj:=wPaper;
    MoveL Offs(pOrigin,248.99,327.71,0.00),v40,fine,tPen\WObj:=wPaper;
    MoveL Offs(pOrigin,248.99,327.71,6.00),v60,z5,tPen\WObj:=wPaper;
    MoveL Offs(pOrigin,247.94,328.76,6.00),vTravel,z5,tPen\WObj:=wPaper;
    MoveL Offs(pOrigin,247.94,328.76,0.00),v60,z0,tPen\WObj:=wPaper;
    MoveL Offs(pOrigin,236.52,340.18,0.00),v40,z0,tPen\WObj:=wPaper;
    MoveL Offs(pOrigin,236.79,340.13,0.00),v40,z0,tPen\WObj:=wPaper;
    MoveL Offs(pOrigin,235.13,338.47,0.00),v40,fine,tPen\WObj:=wPaper;
    MoveL Offs(pOrigin,235.13,338.47,6.00),v60,z5,tPen\WObj:=wPaper;
    MoveL Offs(pOrigin,236.68,337.04,6.00),vTravel,z5,tPen\WObj:=wPaper;
    MoveL Offs(pOrigin,236.68,337.04,0.00),v60,z0,tPen\WObj:=wPaper;
    MoveL Offs(pOrigin,233.23,340.49,0.00),v40,z0,tPen\WObj:=wPaper;
    MoveL Offs(pOrigin,233.94,340.27,0.00),v40,z0,tPen\WObj:=wPaper;
    MoveL Offs(pOrigin,232.44,338.76,0.00),v40,z0,tPen\WObj:=wPaper;
    MoveL Offs(pOrigin,232.63,338.10,0.00),v40,z0,tPen\WObj:=wPaper;
    MoveL Offs(pOrigin,230.53,340.20,0.00),v40,z0,tPen\WObj:=wPaper;
    MoveL Offs(pOrigin,230.95,340.26,0.00),v40,z0,tPen\WObj:=wPaper;
    MoveL Offs(pOrigin,229.14,338.45,0.00),v40,z0,tPen\WObj:=wPaper;
    MoveL Offs(pOrigin,228.32,339.19,0.00),v40,z0,tPen\WObj:=wPaper;
    MoveL Offs(pOrigin,242.56,339.19,0.00),v40,fine,tPen\WObj:=wPaper;
    MoveL Offs(pOrigin,242.56,339.19,6.00),v60,z5,tPen\WObj:=wPaper;
    MoveL Offs(pOrigin,243.83,339.70,6.00),vTravel,z5,tPen\WObj:=wPaper;
    MoveL Offs(pOrigin,243.83,339.70,0.00),v60,z0,tPen\WObj:=wPaper;
    MoveL Offs(pOrigin,240.37,336.24,0.00),v40,z0,tPen\WObj:=wPaper;
    MoveL Offs(pOrigin,241.50,336.02,0.00),v40,z0,tPen\WObj:=wPaper;
    MoveL Offs(pOrigin,243.20,336.02,0.00),v40,z0,tPen\WObj:=wPaper;
    MoveL Offs(pOrigin,243.20,336.08,0.00),v40,z0,tPen\WObj:=wPaper;
  ENDPROC

